(* Logix 5000 project; controller ABB_Drive_Test vendor 1 type 14 code 149 rev 33.12; software revision 33.01 *)

TASK MainTask (continuous, watchdog 500 ms) : T000_MainProgram, CSVProgram, CF_FunctionsProgram

MODULES
   Local : vendor 1 type 14 code 149 (Compact 0, rev 33.12)
      Module_Hart : vendor 58 type 10 code 4 (Compact 2, rev 3.1, Output RPI 80 ms)
      Discrete_IO : Embedded (Compact 1, rev 3.1, Output RPI 20 ms)
      ABBDrive : ETHERNET-MODULE (Ethernet 192.168.2.9, rev 1.1, Output RPI 20 ms)
           ABBDrive:I.Data[0]   // Logic Status Word
           ABBDrive:I.Data[1]   // RPM Actual (INT)
           ABBDrive:I.Data[2]   // DL 1 (Real)
           ABBDrive:I.Data[3]   // DL 1 (Real)
END_MODULES

TYPE ABB_Read :   // Datalinks de Lectura
STRUCT
   Logic_Status_Word : LSW;
   RPM_Feedback : INT;   // RPM Tomada del VSD
   RPM_Referencia : INT;   // Referencia RPM Inyectada
   Output_Power : REAL;
   BusDC : REAL;
   Output_Current : REAL;
   Output_Voltage : REAL;
   PF : REAL;   // Factor de Potencia
   Latest_Fault : INT;
   Accel : BOOL;   // Estado VSD si esta Acelerando
   Descell : BOOL;   // Estado VSD si esta Deshacelerando
END_STRUCT
END_TYPE

TYPE ABB_Write :
STRUCT
   RPM_Reference : INT;
   Run_Forward : BOOL;
   Run_Reverse : BOOL;
   Reset_Fault : BOOL;
END_STRUCT
END_TYPE

TYPE CF_functions :
STRUCT
   command : DINT;   // 1=clear 2=read 3=write 4=append 5=delete 6=rename 7=create dir 8=list 9=list+ 10=list dir 11=detect card 12=get timestamp
   index : DINT;
   offset : DINT;
   REQ_length : DINT;
   DN_length : DINT;
   result : DINT;
   name : STRING;
   newname : STRING;
   data : SINT[460];
   strings : STRING[100];
END_STRUCT
END_TYPE

TYPE ComandVSD :   // Comandos de funcionamiento VSD
STRUCT
   start : BOOL;   // arranque
   stop : BOOL;   // Parada
   reset : BOOL;   // reset VSD
   referencia : REAL;   // Referencia en RPM para VSD AFE
   direction : BOOL;   // Fordware o Reverse
END_STRUCT
END_TYPE

TYPE DateTime :
STRUCT
   year : DINT;
   month : DINT;
   day : DINT;
   hour : DINT;
   minute : DINT;
   second : DINT;
   usec : DINT;
END_STRUCT
END_TYPE

TYPE Dinagrama :   // Estructura de Dinagrama para lectura del SWC PRO
STRUCT
   indiceAux : INT;   // Indice Auxiliar para lectura PLC a SWC
   indice : INT;   // Indice para la lectura del Vector de Potencia
   CT : REAL;   // Valor de la CT para enviar por comunicación a SWC
   PotenciaC : REAL;   // Potencia Cableada valor
   Potencia : REAL;   // Valor de Potencia Actual adquirida por comunicación
   numeroMuestras : INT;   // Numero de Muestras del Stroke de Potencia
   pausa : BOOL;   // Pausa en la adquisión del stroke de potencia
   tiempoMuestreo : INT;   // Tiempo de Muestreo de la señal en ms
   tiempoPausa : INT;   // Tiempo de Pausa para la adquisión de la señal
   vsdActive : BOOL;   // Variador en Referencia
   proximetro : BOOL;   // Señal digital del proximetro tomada de la R003_IO
   inicio : BOOL;   // Inicio para la adquisión de dinagrama, teniendo presente si llego a referencia y demás
   Posicion : REAL;   // Posicion SRP
   Carga : REAL;   // Carga de Sarta Entrada Analoga
   confPos : fuenteEntradaAnaloga;   // Configuracion de Entrada Analoga de posicion
   confCarga : fuenteEntradaAnaloga;   // Configuracion de entrada analoga de carga
   confPot : fuenteEntradaAnaloga;   // Configuracion de entrada analoga VSD
   confCT : fuenteEntradaAnaloga;   // Configuración de Entrada CT
END_STRUCT
END_TYPE

TYPE ethImplicitRead :   // Comunicación para la lectura de los parametros del VSD por ethernet IP
STRUCT
   Enabled : BOOL;   // habilitar Comunicación
   Done : BOOL;   // Se realizó correctamente
   Error : BOOL;   // Se tiene un error en la lectura de los parámetros
   Value : DINT;   // Valor Obtenido
   instance : DINT;   // instancia del parametro
   atribute : INT;   // Atributo del parametro
END_STRUCT
END_TYPE

TYPE ethImplicitWrite :   // Comunicación Para enviar parametros al sistema
STRUCT
   Enabled : BOOL;   // Habilitar
   Done : BOOL;   // Se realizo exitozamente
   ERR : BOOL;   // Error en el envio de la información
   Value : DINT;   // Valor a ingresar
   Instance : DINT;   // Valor de la Instancia
   Atribute : INT;   // Valor del Atributo de la instancia
   clase : INT;
END_STRUCT
END_TYPE

TYPE fuenteEntradaAnaloga :   // Definición de Entrada Analoga ,Fuente de la señal ,rango minimo y maximo
STRUCT
   fuente : INT;   // Canal por el cual se suministra la señal
   Valor : REAL;   // Valor Actual de la señal
   min : REAL;
   max : REAL;
   ValorMinAmp : REAL;
END_STRUCT
END_TYPE

TYPE LSW :   // Drive - Logic Status Word
STRUCT
   Faulted : BOOL;
   Warning : BOOL;
   RunForward : BOOL;
   RunReverse : BOOL;
   Ready : BOOL;
   RemoteRef : BOOL;
   RemoteCrtl : BOOL;
   AtSpeed : BOOL;
END_STRUCT
END_TYPE

TYPE SWC :   // Comunicación Ethernet con el SWC PRO
STRUCT
   comand : ComandVSD;   // Comandos para VSD
   dinagrama : Dinagrama;   // Valores para adquisión del dinagrama
   entradasDigitales : INT;
   salidasDigitales : INT;
   entradasAnalogas : REAL[4];
   salidasAnalogas : REAL[4];
   ABBRead : ABB_Read;   // Valores de Lectura
   etheWrite : ethImplicitWrite;   // Valores de Escritura Ethernet para VSD
   etheRead : ethImplicitRead;   // Valores de Lectura
END_STRUCT
END_TYPE

ADD_ON_INSTRUCTION CF_big_write   (* revision 1.1 *)
// Revision note:
// only act when triggered
VAR_IN_OUT
   command : DINT; {required}
END_VAR
VAR_INPUT
   array_offset : DINT; {required}
END_VAR
VAR_IN_OUT
   CF_ctrl : CF_functions; {required}
   data : SINT[100]; {required}
END_VAR
VAR_OUTPUT
   busy : BOOL; {access Read Only, visible}
END_VAR
VAR
   arsize : DINT;
   stored_req_length : DINT;
   oneshots : DINT;
   bigwrite : BOOL;
   length_diff : DINT;
   bigread : BOOL;
   BW_active : BOOL;
END_VAR

ROUTINE Logic   (* ladder *)
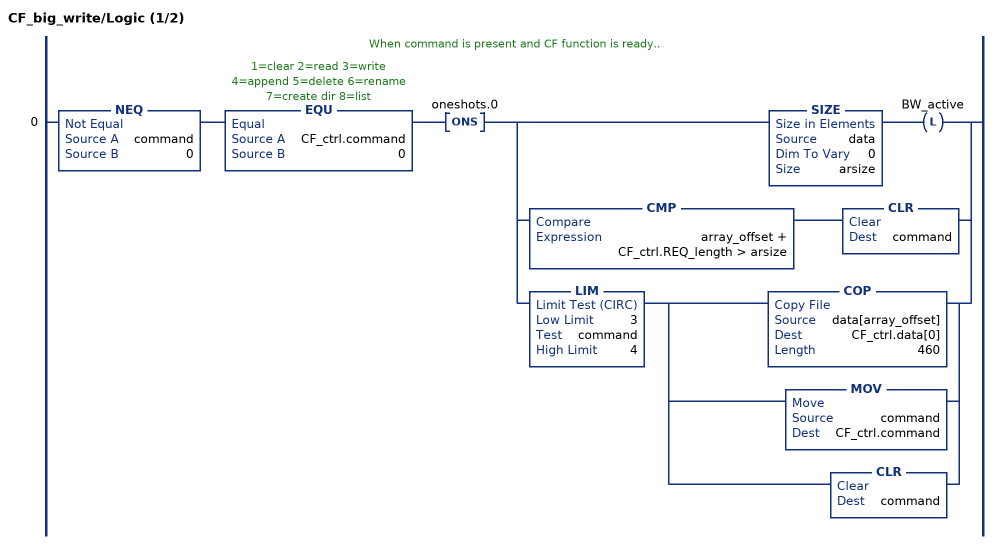
   // When command is present and CF function is ready..
   0: NEQ(command,0)EQU(CF_ctrl.command,0)ONS(oneshots.0)[SIZE(data,0,arsize) OTL(BW_active) ,CMP(array_offset + CF_ctrl.REQ_length > arsize) CLR(command) ,LIM(3,command,4) [COP(data[array_offset],CF_ctrl.data[0],460) ,MOV(command,CF_ctrl.command) ,CLR(command) ] ];
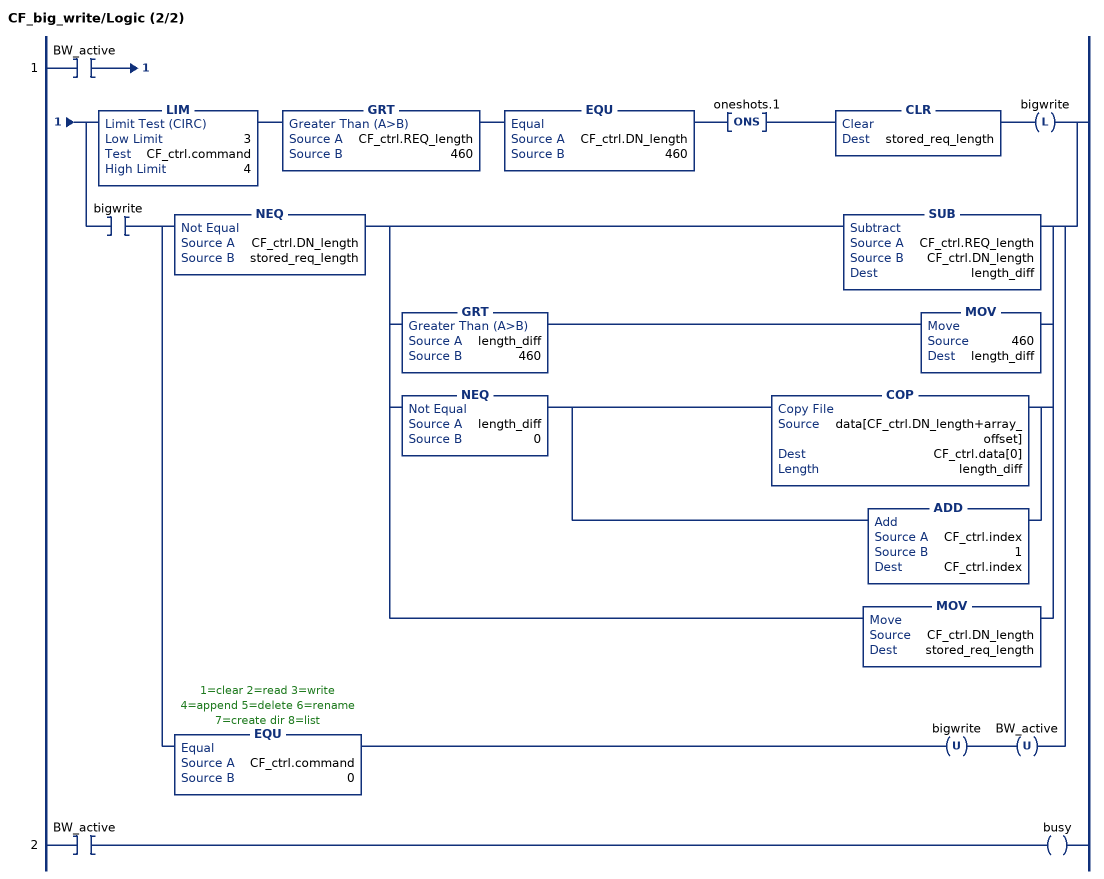
   1: XIC(BW_active)[LIM(3,CF_ctrl.command,4) GRT(CF_ctrl.REQ_length,460) EQU(CF_ctrl.DN_length,460) ONS(oneshots.1) CLR(stored_req_length) OTL(bigwrite) ,XIC(bigwrite) [NEQ(CF_ctrl.DN_length,stored_req_length) [SUB(CF_ctrl.REQ_length,CF_ctrl.DN_length,length_diff) ,GRT(length_diff,460) MOV(460,length_diff) ,NEQ(length_diff,0) [COP(data[CF_ctrl.DN_length+array_offset],CF_ctrl.data[0],length_diff) ,ADD(CF_ctrl.index,1,CF_ctrl.index) ] ,MOV(CF_ctrl.DN_length,stored_req_length) ] ,EQU(CF_ctrl.command,0) OTU(bigwrite) OTU(BW_active) ] ];
   2: XIC(BW_active)OTE(busy);
END_ROUTINE
END_ADD_ON_INSTRUCTION

VAR_GLOBAL   (* controller tags *)
   ABB_GetAtt_Value : DINT := 6000;
   ABB_GetMsg : MESSAGE;
        MessageParameters(ServiceCode := 16#000e, DestinationTag := ABB_GetAtt_Value, ...)
   ABB_Input : ABB_Read := (Logic_Status_Word.Ready := 1, Logic_Status_Word.RemoteRef := 1, Logic_Status_Word.RemoteCrtl := 1, RPM_Referencia := 1440, Output_Power := 5.9449345e-37, BusDC := 678.2, Latest_Fault := 13185);
   ABB_Msg_SetValue : DINT := 1;
   ABB_Output : ABB_Write := (RPM_Reference := 1440);
   ABB_SetMsg : MESSAGE;
        MessageParameters(ServiceCode := 16#0010, LocalElement := ABB_Msg_SetValue, ...)
   asciidata : SINT[11000] := ([0] := 51, [1] := 53, [2] := 56, [3] := 56, [4] := 56, [5] := 44, [6] := 48, [7] := 46, [8] := 48, [9] := 57, [10] := 50, [11] := 55, [12] := 48, [13] := 54, [14] := 54, [15] := 48, [16] := 44, [17] := 50, [18] := 46, [19] := 48, [20] := 48, [21] := 48, [22] := 48, [23] := 48, [24] := 48, [25] := 48, [26] := 48, [27] := 44, [28] := 53, [29] := 46, [30] := 48, [31] := 48, [32] := 48, [33] := 48, [34] := 48, [35] := 48, [36] := 48, [37] := 48, [38] := 44, [39] := 54, [40] := 46, [41] := 48, [42] := 48, [43] := 48, [44] := 48, [45] := 48, [46] := 48, [47] := 48, [48] := 48, [49] := 44, [50] := 55, [51] := 46, [52] := 48, [53] := 48, [54] := 48, [55] := 48, [56] := 48, [57] := 48, [58] := 48, [59] := 48,
        [60] := 44, [61] := 56, [62] := 46, [63] := 48, [64] := 48, [65] := 48, [66] := 48, [67] := 48, [68] := 48, [69] := 48, [70] := 48, [71] := 44, [72] := 57, [73] := 46, [74] := 48, [75] := 48, [76] := 48, [77] := 48, [78] := 48, [79] := 48, [80] := 48, [81] := 48, [82] := 44, [83] := 49, [84] := 48, [85] := 46, [86] := 48, [87] := 48, [88] := 48, [89] := 48, [90] := 48, [91] := 48, [92] := 48, [93] := 44, [94] := 49, [95] := 49, [96] := 46, [97] := 48, [98] := 48, [99] := 48, [100] := 48, [101] := 48, [102] := 48, [103] := 48, [104] := 44, [105] := 49, [106] := 50, [107] := 46, [108] := 48, [109] := 48, [110] := 48, [111] := 48, [112] := 48, [113] := 48, [114] := 48, [115] := 44, [116] := 49, [117] := 46, [118] := 48, [119] := 48,
        [120] := 48, [121] := 48, [122] := 48, [123] := 48, [124] := 48, [125] := 48, [126] := 13, [127] := 10, [128] := 51, [129] := 53, [130] := 56, [131] := 56, [132] := 56, [133] := 44, [134] := 48, [135] := 46, [136] := 48, [137] := 57, [138] := 50, [139] := 55, [140] := 49, [141] := 56, [142] := 49, [143] := 55, [144] := 44, [145] := 50, [146] := 46, [147] := 48, [148] := 48, [149] := 48, [150] := 48, [151] := 48, [152] := 48, [153] := 48, [154] := 48, [155] := 44, [156] := 53, [157] := 46, [158] := 48, [159] := 48, [160] := 48, [161] := 48, [162] := 48, [163] := 48, [164] := 48, [165] := 48, [166] := 44, [167] := 54, [168] := 46, [169] := 48, [170] := 48, [171] := 48, [172] := 48, [173] := 48, [174] := 48, [175] := 48, [176] := 48, [177] := 44, [178] := 55, [179] := 46,
        [180] := 48, [181] := 48, [182] := 48, [183] := 48, [184] := 48, [185] := 48, [186] := 48, [187] := 48, [188] := 44, [189] := 56, [190] := 46, [191] := 48, [192] := 48, [193] := 48, [194] := 48, [195] := 48, [196] := 48, [197] := 48, [198] := 48, [199] := 44, [200] := 57, [201] := 46, [202] := 48, [203] := 48, [204] := 48, [205] := 48, [206] := 48, [207] := 48, [208] := 48, [209] := 48, [210] := 44, [211] := 49, [212] := 48, [213] := 46, [214] := 48, [215] := 48, [216] := 48, [217] := 48, [218] := 48, [219] := 48, [220] := 48, [221] := 44, [222] := 49, [223] := 49, [224] := 46, [225] := 48, [226] := 48, [227] := 48, [228] := 48, [229] := 48, [230] := 48, [231] := 48, [232] := 44, [233] := 49, [234] := 50, [235] := 46, [236] := 48, [237] := 48, [238] := 48, [239] := 48,
        [240] := 48, [241] := 48, [242] := 48, [243] := 44, [244] := 49, [245] := 46, [246] := 48, [247] := 48, [248] := 48, [249] := 48, [250] := 48, [251] := 48, [252] := 48, [253] := 48, [254] := 13, [255] := 10, [256] := 51, [257] := 53, [258] := 56, [259] := 56, [260] := 56, [261] := 44, [262] := 48, [263] := 46, [264] := 48, [265] := 57, [266] := 50, [267] := 55, [268] := 50, [269] := 57, [270] := 55, [271] := 53, [272] := 44, [273] := 50, [274] := 46, [275] := 48, [276] := 48, [277] := 48, [278] := 48, [279] := 48, [280] := 48, [281] := 48, [282] := 48, [283] := 44, [284] := 53, [285] := 46, [286] := 48, [287] := 48, [288] := 48, [289] := 48, [290] := 48, [291] := 48, [292] := 48, [293] := 48, [294] := 44, [295] := 54, [296] := 46, [297] := 48, [298] := 48, [299] := 48,
        [300] := 48, [301] := 48, [302] := 48, [303] := 48, [304] := 48, [305] := 44, [306] := 55, [307] := 46, [308] := 48, [309] := 48, [310] := 48, [311] := 48, [312] := 48, [313] := 48, [314] := 48, [315] := 48, [316] := 44, [317] := 56, [318] := 46, [319] := 48, [320] := 48, [321] := 48, [322] := 48, [323] := 48, [324] := 48, [325] := 48, [326] := 48, [327] := 44, [328] := 57, [329] := 46, [330] := 48, [331] := 48, [332] := 48, [333] := 48, [334] := 48, [335] := 48, [336] := 48, [337] := 48, [338] := 44, [339] := 49, [340] := 48, [341] := 46, [342] := 48, [343] := 48, [344] := 48, [345] := 48, [346] := 48, [347] := 48, [348] := 48, [349] := 44, [350] := 49, [351] := 49, [352] := 46, [353] := 48, [354] := 48, [355] := 48, [356] := 48, [357] := 48, [358] := 48, [359] := 48,
        [360] := 44, [361] := 49, [362] := 50, [363] := 46, [364] := 48, [365] := 48, [366] := 48, [367] := 48, [368] := 48, [369] := 48, [370] := 48, [371] := 44, [372] := 49, [373] := 46, [374] := 48, [375] := 48, [376] := 48, [377] := 48, [378] := 48, [379] := 48, [380] := 48, [381] := 48, [382] := 13, [383] := 10, [384] := 51, [385] := 53, [386] := 56, [387] := 56, [388] := 56, [389] := 44, [390] := 48, [391] := 46, [392] := 48, [393] := 57, [394] := 50, [395] := 55, [396] := 52, [397] := 49, [398] := 51, [399] := 50, [400] := 44, [401] := 50, [402] := 46, [403] := 48, [404] := 48, [405] := 48, [406] := 48, [407] := 48, [408] := 48, [409] := 48, [410] := 48, [411] := 44, [412] := 53, [413] := 46, [414] := 48, [415] := 48, [416] := 48, [417] := 48, [418] := 48, [419] := 48,
        [420] := 48, [421] := 48, [422] := 44, [423] := 54, [424] := 46, [425] := 48, [426] := 48, [427] := 48, [428] := 48, [429] := 48, [430] := 48, [431] := 48, [432] := 48, [433] := 44, [434] := 55, [435] := 46, [436] := 48, [437] := 48, [438] := 48, [439] := 48, [440] := 48, [441] := 48, [442] := 48, [443] := 48, [444] := 44, [445] := 56, [446] := 46, [447] := 48, [448] := 48, [449] := 48, [450] := 48, [451] := 48, [452] := 48, [453] := 48, [454] := 48, [455] := 44, [456] := 57, [457] := 46, [458] := 48, [459] := 48, [460] := 48, [461] := 48, [462] := 48, [463] := 48, [464] := 48, [465] := 48, [466] := 44, [467] := 49, [468] := 48, [469] := 46, [470] := 48, [471] := 48, [472] := 48, [473] := 48, [474] := 48, [475] := 48, [476] := 48, [477] := 44, [478] := 49, [479] := 49,
        [480] := 46, [481] := 48, [482] := 48, [483] := 48, [484] := 48, [485] := 48, [486] := 48, [487] := 48, [488] := 44, [489] := 49, [490] := 50, [491] := 46, [492] := 48, [493] := 48, [494] := 48, [495] := 48, [496] := 48, [497] := 48, [498] := 48, [499] := 44, [500] := 49, [501] := 46, [502] := 48, [503] := 48, [504] := 48, [505] := 48, [506] := 48, [507] := 48, [508] := 48, [509] := 48, [510] := 13, [511] := 10, [512] := 51, [513] := 53, [514] := 56, [515] := 56, [516] := 56, [517] := 44, [518] := 48, [519] := 46, [520] := 48, [521] := 57, [522] := 50, [523] := 55, [524] := 53, [525] := 50, [526] := 57, [527] := 48, [528] := 44, [529] := 50, [530] := 46, [531] := 48, [532] := 48, [533] := 48, [534] := 48, [535] := 48, [536] := 48, [537] := 48, [538] := 48, [539] := 44,
        [540] := 53, [541] := 46, [542] := 48, [543] := 48, [544] := 48, [545] := 48, [546] := 48, [547] := 48, [548] := 48, [549] := 48, [550] := 44, [551] := 54, [552] := 46, [553] := 48, [554] := 48, [555] := 48, [556] := 48, [557] := 48, [558] := 48, [559] := 48, [560] := 48, [561] := 44, [562] := 55, [563] := 46, [564] := 48, [565] := 48, [566] := 48, [567] := 48, [568] := 48, [569] := 48, [570] := 48, [571] := 48, [572] := 44, [573] := 56, [574] := 46, [575] := 48, [576] := 48, [577] := 48, [578] := 48, [579] := 48, [580] := 48, [581] := 48, [582] := 48, [583] := 44, [584] := 57, [585] := 46, [586] := 48, [587] := 48, [588] := 48, [589] := 48, [590] := 48, [591] := 48, [592] := 48, [593] := 48, [594] := 44, [595] := 49, [596] := 48, [597] := 46, [598] := 48, [599] := 48,
        [600] := 48, [601] := 48, [602] := 48, [603] := 48, [604] := 48, [605] := 44, [606] := 49, [607] := 49, [608] := 46, [609] := 48, [610] := 48, [611] := 48, [612] := 48, [613] := 48, [614] := 48, [615] := 48, [616] := 44, [617] := 49, [618] := 50, [619] := 46, [620] := 48, [621] := 48, [622] := 48, [623] := 48, [624] := 48, [625] := 48, [626] := 48, [627] := 44, [628] := 49, [629] := 46, [630] := 48, [631] := 48, [632] := 48, [633] := 48, [634] := 48, [635] := 48, [636] := 48, [637] := 48, [638] := 13, [639] := 10, [640] := 51, [641] := 53, [642] := 56, [643] := 56, [644] := 56, [645] := 44, [646] := 48, [647] := 46, [648] := 48, [649] := 57, [650] := 50, [651] := 55, [652] := 54, [653] := 52, [654] := 52, [655] := 55, [656] := 44, [657] := 50, [658] := 46, [659] := 48,
        [660] := 48, [661] := 48, [662] := 48, [663] := 48, [664] := 48, [665] := 48, [666] := 48, [667] := 44, [668] := 53, [669] := 46, [670] := 48, [671] := 48, [672] := 48, [673] := 48, [674] := 48, [675] := 48, [676] := 48, [677] := 48, [678] := 44, [679] := 54, [680] := 46, [681] := 48, [682] := 48, [683] := 48, [684] := 48, [685] := 48, [686] := 48, [687] := 48, [688] := 48, [689] := 44, [690] := 55, [691] := 46, [692] := 48, [693] := 48, [694] := 48, [695] := 48, [696] := 48, [697] := 48, [698] := 48, [699] := 48, [700] := 44, [701] := 56, [702] := 46, [703] := 48, [704] := 48, [705] := 48, [706] := 48, [707] := 48, [708] := 48, [709] := 48, [710] := 48, [711] := 44, [712] := 57, [713] := 46, [714] := 48, [715] := 48, [716] := 48, [717] := 48, [718] := 48, [719] := 48,
        [720] := 48, [721] := 48, [722] := 44, [723] := 49, [724] := 48, [725] := 46, [726] := 48, [727] := 48, [728] := 48, [729] := 48, [730] := 48, [731] := 48, [732] := 48, [733] := 44, [734] := 49, [735] := 49, [736] := 46, [737] := 48, [738] := 48, [739] := 48, [740] := 48, [741] := 48, [742] := 48, [743] := 48, [744] := 44, [745] := 49, [746] := 50, [747] := 46, [748] := 48, [749] := 48, [750] := 48, [751] := 48, [752] := 48, [753] := 48, [754] := 48, [755] := 44, [756] := 49, [757] := 46, [758] := 48, [759] := 48, [760] := 48, [761] := 48, [762] := 48, [763] := 48, [764] := 48, [765] := 48, [766] := 13, [767] := 10, [768] := 51, [769] := 53, [770] := 56, [771] := 56, [772] := 56, [773] := 44, [774] := 48, [775] := 46, [776] := 48, [777] := 57, [778] := 50, [779] := 55,
        [780] := 55, [781] := 54, [782] := 48, [783] := 53, [784] := 44, [785] := 50, [786] := 46, [787] := 48, [788] := 48, [789] := 48, [790] := 48, [791] := 48, [792] := 48, [793] := 48, [794] := 48, [795] := 44, [796] := 53, [797] := 46, [798] := 48, [799] := 48, [800] := 48, [801] := 48, [802] := 48, [803] := 48, [804] := 48, [805] := 48, [806] := 44, [807] := 54, [808] := 46, [809] := 48, [810] := 48, [811] := 48, [812] := 48, [813] := 48, [814] := 48, [815] := 48, [816] := 48, [817] := 44, [818] := 55, [819] := 46, [820] := 48, [821] := 48, [822] := 48, [823] := 48, [824] := 48, [825] := 48, [826] := 48, [827] := 48, [828] := 44, [829] := 56, [830] := 46, [831] := 48, [832] := 48, [833] := 48, [834] := 48, [835] := 48, [836] := 48, [837] := 48, [838] := 48, [839] := 44,
        [840] := 57, [841] := 46, [842] := 48, [843] := 48, [844] := 48, [845] := 48, [846] := 48, [847] := 48, [848] := 48, [849] := 48, [850] := 44, [851] := 49, [852] := 48, [853] := 46, [854] := 48, [855] := 48, [856] := 48, [857] := 48, [858] := 48, [859] := 48, [860] := 48, [861] := 44, [862] := 49, [863] := 49, [864] := 46, [865] := 48, [866] := 48, [867] := 48, [868] := 48, [869] := 48, [870] := 48, [871] := 48, [872] := 44, [873] := 49, [874] := 50, [875] := 46, [876] := 48, [877] := 48, [878] := 48, [879] := 48, [880] := 48, [881] := 48, [882] := 48, [883] := 44, [884] := 49, [885] := 46, [886] := 48, [887] := 48, [888] := 48, [889] := 48, [890] := 48, [891] := 48, [892] := 48, [893] := 48, [894] := 13, [895] := 10, [896] := 51, [897] := 53, [898] := 56, [899] := 56,
        [900] := 56, [901] := 44, [902] := 48, [903] := 46, [904] := 48, [905] := 57, [906] := 50, [907] := 55, [908] := 56, [909] := 55, [910] := 54, [911] := 50, [912] := 44, [913] := 50, [914] := 46, [915] := 48, [916] := 48, [917] := 48, [918] := 48, [919] := 48, [920] := 48, [921] := 48, [922] := 48, [923] := 44, [924] := 53, [925] := 46, [926] := 48, [927] := 48, [928] := 48, [929] := 48, [930] := 48, [931] := 48, [932] := 48, [933] := 48, [934] := 44, [935] := 54, [936] := 46, [937] := 48, [938] := 48, [939] := 48, [940] := 48, [941] := 48, [942] := 48, [943] := 48, [944] := 48, [945] := 44, [946] := 55, [947] := 46, [948] := 48, [949] := 48, [950] := 48, [951] := 48, [952] := 48, [953] := 48, [954] := 48, [955] := 48, [956] := 44, [957] := 56, [958] := 46, [959] := 48,
        [960] := 48, [961] := 48, [962] := 48, [963] := 48, [964] := 48, [965] := 48, [966] := 48, [967] := 44, [968] := 57, [969] := 46, [970] := 48, [971] := 48, [972] := 48, [973] := 48, [974] := 48, [975] := 48, [976] := 48, [977] := 48, [978] := 44, [979] := 49, [980] := 48, [981] := 46, [982] := 48, [983] := 48, [984] := 48, [985] := 48, [986] := 48, [987] := 48, [988] := 48, [989] := 44, [990] := 49, [991] := 49, [992] := 46, [993] := 48, [994] := 48, [995] := 48, [996] := 48, [997] := 48, [998] := 48, [999] := 48, [1000] := 44, [1001] := 49, [1002] := 50, [1003] := 46, [1004] := 48, [1005] := 48, [1006] := 48, [1007] := 48, [1008] := 48, [1009] := 48, [1010] := 48, [1011] := 44, [1012] := 49, [1013] := 46, [1014] := 48, [1015] := 48, [1016] := 48, [1017] := 48, [1018] := 48, [1019] := 48,
        [1020] := 48, [1021] := 48, [1022] := 13, [1023] := 10, [1024] := 51, [1025] := 53, [1026] := 56, [1027] := 56, [1028] := 56, [1029] := 44, [1030] := 48, [1031] := 46, [1032] := 48, [1033] := 57, [1034] := 50, [1035] := 55, [1036] := 57, [1037] := 57, [1038] := 49, [1039] := 57, [1040] := 44, [1041] := 50, [1042] := 46, [1043] := 48, [1044] := 48, [1045] := 48, [1046] := 48, [1047] := 48, [1048] := 48, [1049] := 48, [1050] := 48, [1051] := 44, [1052] := 53, [1053] := 46, [1054] := 48, [1055] := 48, [1056] := 48, [1057] := 48, [1058] := 48, [1059] := 48, [1060] := 48, [1061] := 48, [1062] := 44, [1063] := 54, [1064] := 46, [1065] := 48, [1066] := 48, [1067] := 48, [1068] := 48, [1069] := 48, [1070] := 48, [1071] := 48, [1072] := 48, [1073] := 44, [1074] := 55, [1075] := 46, [1076] := 48, [1077] := 48, [1078] := 48, [1079] := 48,
        [1080] := 48, [1081] := 48, [1082] := 48, [1083] := 48, [1084] := 44, [1085] := 56, [1086] := 46, [1087] := 48, [1088] := 48, [1089] := 48, [1090] := 48, [1091] := 48, [1092] := 48, [1093] := 48, [1094] := 48, [1095] := 44, [1096] := 57, [1097] := 46, [1098] := 48, [1099] := 48, [1100] := 48, [1101] := 48, [1102] := 48, [1103] := 48, [1104] := 48, [1105] := 48, [1106] := 44, [1107] := 49, [1108] := 48, [1109] := 46, [1110] := 48, [1111] := 48, [1112] := 48, [1113] := 48, [1114] := 48, [1115] := 48, [1116] := 48, [1117] := 44, [1118] := 49, [1119] := 49, [1120] := 46, [1121] := 48, [1122] := 48, [1123] := 48, [1124] := 48, [1125] := 48, [1126] := 48, [1127] := 48, [1128] := 44, [1129] := 49, [1130] := 50, [1131] := 46, [1132] := 48, [1133] := 48, [1134] := 48, [1135] := 48, [1136] := 48, [1137] := 48, [1138] := 48, [1139] := 44,
        [1140] := 49, [1141] := 46, [1142] := 48, [1143] := 48, [1144] := 48, [1145] := 48, [1146] := 48, [1147] := 48, [1148] := 48, [1149] := 48, [1150] := 13, [1151] := 10, [1152] := 51, [1153] := 53, [1154] := 56, [1155] := 56, [1156] := 56, [1157] := 44, [1158] := 48, [1159] := 46, [1160] := 48, [1161] := 57, [1162] := 50, [1163] := 56, [1164] := 49, [1165] := 48, [1166] := 55, [1167] := 54, [1168] := 44, [1169] := 50, [1170] := 46, [1171] := 48, [1172] := 48, [1173] := 48, [1174] := 48, [1175] := 48, [1176] := 48, [1177] := 48, [1178] := 48, [1179] := 44, [1180] := 53, [1181] := 46, [1182] := 48, [1183] := 48, [1184] := 48, [1185] := 48, [1186] := 48, [1187] := 48, [1188] := 48, [1189] := 48, [1190] := 44, [1191] := 54, [1192] := 46, [1193] := 48, [1194] := 48, [1195] := 48, [1196] := 48, [1197] := 48, [1198] := 48, [1199] := 48,
        [1200] := 48, [1201] := 44, [1202] := 55, [1203] := 46, [1204] := 48, [1205] := 48, [1206] := 48, [1207] := 48, [1208] := 48, [1209] := 48, [1210] := 48, [1211] := 48, [1212] := 44, [1213] := 56, [1214] := 46, [1215] := 48, [1216] := 48, [1217] := 48, [1218] := 48, [1219] := 48, [1220] := 48, [1221] := 48, [1222] := 48, [1223] := 44, [1224] := 57, [1225] := 46, [1226] := 48, [1227] := 48, [1228] := 48, [1229] := 48, [1230] := 48, [1231] := 48, [1232] := 48, [1233] := 48, [1234] := 44, [1235] := 49, [1236] := 48, [1237] := 46, [1238] := 48, [1239] := 48, [1240] := 48, [1241] := 48, [1242] := 48, [1243] := 48, [1244] := 48, [1245] := 44, [1246] := 49, [1247] := 49, [1248] := 46, [1249] := 48, [1250] := 48, [1251] := 48, [1252] := 48, [1253] := 48, [1254] := 48, [1255] := 48, [1256] := 44, [1257] := 49, [1258] := 50, [1259] := 46,
        [1260] := 48, [1261] := 48, [1262] := 48, [1263] := 48, [1264] := 48, [1265] := 48, [1266] := 48, [1267] := 44, [1268] := 49, [1269] := 46, [1270] := 48, [1271] := 48, [1272] := 48, [1273] := 48, [1274] := 48, [1275] := 48, [1276] := 48, [1277] := 48, [1278] := 13, [1279] := 10, [1280] := 51, [1281] := 53, [1282] := 56, [1283] := 56, [1284] := 56, [1285] := 44, [1286] := 48, [1287] := 46, [1288] := 48, [1289] := 57, [1290] := 50, [1291] := 56, [1292] := 50, [1293] := 50, [1294] := 51, [1295] := 52, [1296] := 44, [1297] := 50, [1298] := 46, [1299] := 48, [1300] := 48, [1301] := 48, [1302] := 48, [1303] := 48, [1304] := 48, [1305] := 48, [1306] := 48, [1307] := 44, [1308] := 53, [1309] := 46, [1310] := 48, [1311] := 48, [1312] := 48, [1313] := 48, [1314] := 48, [1315] := 48, [1316] := 48, [1317] := 48, [1318] := 44, [1319] := 54,
        [1320] := 46, [1321] := 48, [1322] := 48, [1323] := 48, [1324] := 48, [1325] := 48, [1326] := 48, [1327] := 48, [1328] := 48, [1329] := 44, [1330] := 55, [1331] := 46, [1332] := 48, [1333] := 48, [1334] := 48, [1335] := 48, [1336] := 48, [1337] := 48, [1338] := 48, [1339] := 48, [1340] := 44, [1341] := 56, [1342] := 46, [1343] := 48, [1344] := 48, [1345] := 48, [1346] := 48, [1347] := 48, [1348] := 48, [1349] := 48, [1350] := 48, [1351] := 44, [1352] := 57, [1353] := 46, [1354] := 48, [1355] := 48, [1356] := 48, [1357] := 48, [1358] := 48, [1359] := 48, [1360] := 48, [1361] := 48, [1362] := 44, [1363] := 49, [1364] := 48, [1365] := 46, [1366] := 48, [1367] := 48, [1368] := 48, [1369] := 48, [1370] := 48, [1371] := 48, [1372] := 48, [1373] := 44, [1374] := 49, [1375] := 49, [1376] := 46, [1377] := 48, [1378] := 48, [1379] := 48,
        [1380] := 48, [1381] := 48, [1382] := 48, [1383] := 48, [1384] := 44, [1385] := 49, [1386] := 50, [1387] := 46, [1388] := 48, [1389] := 48, [1390] := 48, [1391] := 48, [1392] := 48, [1393] := 48, [1394] := 48, [1395] := 44, [1396] := 49, [1397] := 46, [1398] := 48, [1399] := 48, [1400] := 48, [1401] := 48, [1402] := 48, [1403] := 48, [1404] := 48, [1405] := 48, [1406] := 13, [1407] := 10, [1408] := 51, [1409] := 53, [1410] := 56, [1411] := 56, [1412] := 56, [1413] := 44, [1414] := 48, [1415] := 46, [1416] := 48, [1417] := 57, [1418] := 50, [1419] := 56, [1420] := 51, [1421] := 51, [1422] := 57, [1423] := 49, [1424] := 44, [1425] := 50, [1426] := 46, [1427] := 48, [1428] := 48, [1429] := 48, [1430] := 48, [1431] := 48, [1432] := 48, [1433] := 48, [1434] := 48, [1435] := 44, [1436] := 53, [1437] := 46, [1438] := 48, [1439] := 48,
        [1440] := 48, [1441] := 48, [1442] := 48, [1443] := 48, [1444] := 48, [1445] := 48, [1446] := 44, [1447] := 54, [1448] := 46, [1449] := 48, [1450] := 48, [1451] := 48, [1452] := 48, [1453] := 48, [1454] := 48, [1455] := 48, [1456] := 48, [1457] := 44, [1458] := 55, [1459] := 46, [1460] := 48, [1461] := 48, [1462] := 48, [1463] := 48, [1464] := 48, [1465] := 48, [1466] := 48, [1467] := 48, [1468] := 44, [1469] := 56, [1470] := 46, [1471] := 48, [1472] := 48, [1473] := 48, [1474] := 48, [1475] := 48, [1476] := 48, [1477] := 48, [1478] := 48, [1479] := 44, [1480] := 57, [1481] := 46, [1482] := 48, [1483] := 48, [1484] := 48, [1485] := 48, [1486] := 48, [1487] := 48, [1488] := 48, [1489] := 48, [1490] := 44, [1491] := 49, [1492] := 48, [1493] := 46, [1494] := 48, [1495] := 48, [1496] := 48, [1497] := 48, [1498] := 48, [1499] := 48,
        [1500] := 48, [1501] := 44, [1502] := 49, [1503] := 49, [1504] := 46, [1505] := 48, [1506] := 48, [1507] := 48, [1508] := 48, [1509] := 48, [1510] := 48, [1511] := 48, [1512] := 44, [1513] := 49, [1514] := 50, [1515] := 46, [1516] := 48, [1517] := 48, [1518] := 48, [1519] := 48, [1520] := 48, [1521] := 48, [1522] := 48, [1523] := 44, [1524] := 49, [1525] := 46, [1526] := 48, [1527] := 48, [1528] := 48, [1529] := 48, [1530] := 48, [1531] := 48, [1532] := 48, [1533] := 48, [1534] := 13, [1535] := 10, [1536] := 51, [1537] := 53, [1538] := 56, [1539] := 56, [1540] := 56, [1541] := 44, [1542] := 48, [1543] := 46, [1544] := 48, [1545] := 57, [1546] := 50, [1547] := 56, [1548] := 52, [1549] := 53, [1550] := 52, [1551] := 56, [1552] := 44, [1553] := 50, [1554] := 46, [1555] := 48, [1556] := 48, [1557] := 48, [1558] := 48, [1559] := 48,
        [1560] := 48, [1561] := 48, [1562] := 48, [1563] := 44, [1564] := 53, [1565] := 46, [1566] := 48, [1567] := 48, [1568] := 48, [1569] := 48, [1570] := 48, [1571] := 48, [1572] := 48, [1573] := 48, [1574] := 44, [1575] := 54, [1576] := 46, [1577] := 48, [1578] := 48, [1579] := 48, [1580] := 48, [1581] := 48, [1582] := 48, [1583] := 48, [1584] := 48, [1585] := 44, [1586] := 55, [1587] := 46, [1588] := 48, [1589] := 48, [1590] := 48, [1591] := 48, [1592] := 48, [1593] := 48, [1594] := 48, [1595] := 48, [1596] := 44, [1597] := 56, [1598] := 46, [1599] := 48, [1600] := 48, [1601] := 48, [1602] := 48, [1603] := 48, [1604] := 48, [1605] := 48, [1606] := 48, [1607] := 44, [1608] := 57, [1609] := 46, [1610] := 48, [1611] := 48, [1612] := 48, [1613] := 48, [1614] := 48, [1615] := 48, [1616] := 48, [1617] := 48, [1618] := 44, [1619] := 49,
        [1620] := 48, [1621] := 46, [1622] := 48, [1623] := 48, [1624] := 48, [1625] := 48, [1626] := 48, [1627] := 48, [1628] := 48, [1629] := 44, [1630] := 49, [1631] := 49, [1632] := 46, [1633] := 48, [1634] := 48, [1635] := 48, [1636] := 48, [1637] := 48, [1638] := 48, [1639] := 48, [1640] := 44, [1641] := 49, [1642] := 50, [1643] := 46, [1644] := 48, [1645] := 48, [1646] := 48, [1647] := 48, [1648] := 48, [1649] := 48, [1650] := 48, [1651] := 44, [1652] := 49, [1653] := 46, [1654] := 48, [1655] := 48, [1656] := 48, [1657] := 48, [1658] := 48, [1659] := 48, [1660] := 48, [1661] := 48, [1662] := 13, [1663] := 10, [1664] := 51, [1665] := 53, [1666] := 56, [1667] := 56, [1668] := 56, [1669] := 44, [1670] := 48, [1671] := 46, [1672] := 48, [1673] := 57, [1674] := 50, [1675] := 56, [1676] := 53, [1677] := 55, [1678] := 48, [1679] := 54,
        [1680] := 44, [1681] := 50, [1682] := 46, [1683] := 48, [1684] := 48, [1685] := 48, [1686] := 48, [1687] := 48, [1688] := 48, [1689] := 48, [1690] := 48, [1691] := 44, [1692] := 53, [1693] := 46, [1694] := 48, [1695] := 48, [1696] := 48, [1697] := 48, [1698] := 48, [1699] := 48, [1700] := 48, [1701] := 48, [1702] := 44, [1703] := 54, [1704] := 46, [1705] := 48, [1706] := 48, [1707] := 48, [1708] := 48, [1709] := 48, [1710] := 48, [1711] := 48, [1712] := 48, [1713] := 44, [1714] := 55, [1715] := 46, [1716] := 48, [1717] := 48, [1718] := 48, [1719] := 48, [1720] := 48, [1721] := 48, [1722] := 48, [1723] := 48, [1724] := 44, [1725] := 56, [1726] := 46, [1727] := 48, [1728] := 48, [1729] := 48, [1730] := 48, [1731] := 48, [1732] := 48, [1733] := 48, [1734] := 48, [1735] := 44, [1736] := 57, [1737] := 46, [1738] := 48, [1739] := 48,
        [1740] := 48, [1741] := 48, [1742] := 48, [1743] := 48, [1744] := 48, [1745] := 48, [1746] := 44, [1747] := 49, [1748] := 48, [1749] := 46, [1750] := 48, [1751] := 48, [1752] := 48, [1753] := 48, [1754] := 48, [1755] := 48, [1756] := 48, [1757] := 44, [1758] := 49, [1759] := 49, [1760] := 46, [1761] := 48, [1762] := 48, [1763] := 48, [1764] := 48, [1765] := 48, [1766] := 48, [1767] := 48, [1768] := 44, [1769] := 49, [1770] := 50, [1771] := 46, [1772] := 48, [1773] := 48, [1774] := 48, [1775] := 48, [1776] := 48, [1777] := 48, [1778] := 48, [1779] := 44, [1780] := 49, [1781] := 46, [1782] := 48, [1783] := 48, [1784] := 48, [1785] := 48, [1786] := 48, [1787] := 48, [1788] := 48, [1789] := 48, [1790] := 13, [1791] := 10, [1792] := 51, [1793] := 53, [1794] := 56, [1795] := 56, [1796] := 56, [1797] := 44, [1798] := 48, [1799] := 46,
        [1800] := 48, [1801] := 57, [1802] := 50, [1803] := 56, [1804] := 54, [1805] := 56, [1806] := 54, [1807] := 51, [1808] := 44, [1809] := 50, [1810] := 46, [1811] := 48, [1812] := 48, [1813] := 48, [1814] := 48, [1815] := 48, [1816] := 48, [1817] := 48, [1818] := 48, [1819] := 44, [1820] := 53, [1821] := 46, [1822] := 48, [1823] := 48, [1824] := 48, [1825] := 48, [1826] := 48, [1827] := 48, [1828] := 48, [1829] := 48, [1830] := 44, [1831] := 54, [1832] := 46, [1833] := 48, [1834] := 48, [1835] := 48, [1836] := 48, [1837] := 48, [1838] := 48, [1839] := 48, [1840] := 48, [1841] := 44, [1842] := 55, [1843] := 46, [1844] := 48, [1845] := 48, [1846] := 48, [1847] := 48, [1848] := 48, [1849] := 48, [1850] := 48, [1851] := 48, [1852] := 44, [1853] := 56, [1854] := 46, [1855] := 48, [1856] := 48, [1857] := 48, [1858] := 48, [1859] := 48,
        [1860] := 48, [1861] := 48, [1862] := 48, [1863] := 44, [1864] := 57, [1865] := 46, [1866] := 48, [1867] := 48, [1868] := 48, [1869] := 48, [1870] := 48, [1871] := 48, [1872] := 48, [1873] := 48, [1874] := 44, [1875] := 49, [1876] := 48, [1877] := 46, [1878] := 48, [1879] := 48, [1880] := 48, [1881] := 48, [1882] := 48, [1883] := 48, [1884] := 48, [1885] := 44, [1886] := 49, [1887] := 49, [1888] := 46, [1889] := 48, [1890] := 48, [1891] := 48, [1892] := 48, [1893] := 48, [1894] := 48, [1895] := 48, [1896] := 44, [1897] := 49, [1898] := 50, [1899] := 46, [1900] := 48, [1901] := 48, [1902] := 48, [1903] := 48, [1904] := 48, [1905] := 48, [1906] := 48, [1907] := 44, [1908] := 49, [1909] := 46, [1910] := 48, [1911] := 48, [1912] := 48, [1913] := 48, [1914] := 48, [1915] := 48, [1916] := 48, [1917] := 48, [1918] := 13, [1919] := 10,
        [1920] := 51, [1921] := 53, [1922] := 56, [1923] := 56, [1924] := 56, [1925] := 44, [1926] := 48, [1927] := 46, [1928] := 48, [1929] := 57, [1930] := 50, [1931] := 56, [1932] := 56, [1933] := 48, [1934] := 50, [1935] := 49, [1936] := 44, [1937] := 50, [1938] := 46, [1939] := 48, [1940] := 48, [1941] := 48, [1942] := 48, [1943] := 48, [1944] := 48, [1945] := 48, [1946] := 48, [1947] := 44, [1948] := 53, [1949] := 46, [1950] := 48, [1951] := 48, [1952] := 48, [1953] := 48, [1954] := 48, [1955] := 48, [1956] := 48, [1957] := 48, [1958] := 44, [1959] := 54, [1960] := 46, [1961] := 48, [1962] := 48, [1963] := 48, [1964] := 48, [1965] := 48, [1966] := 48, [1967] := 48, [1968] := 48, [1969] := 44, [1970] := 55, [1971] := 46, [1972] := 48, [1973] := 48, [1974] := 48, [1975] := 48, [1976] := 48, [1977] := 48, [1978] := 48, [1979] := 48,
        [1980] := 44, [1981] := 56, [1982] := 46, [1983] := 48, [1984] := 48, [1985] := 48, [1986] := 48, [1987] := 48, [1988] := 48, [1989] := 48, [1990] := 48, [1991] := 44, [1992] := 57, [1993] := 46, [1994] := 48, [1995] := 48, [1996] := 48, [1997] := 48, [1998] := 48, [1999] := 48, [2000] := 48, [2001] := 48, [2002] := 44, [2003] := 49, [2004] := 48, [2005] := 46, [2006] := 48, [2007] := 48, [2008] := 48, [2009] := 48, [2010] := 48, [2011] := 48, [2012] := 48, [2013] := 44, [2014] := 49, [2015] := 49, [2016] := 46, [2017] := 48, [2018] := 48, [2019] := 48, [2020] := 48, [2021] := 48, [2022] := 48, [2023] := 48, [2024] := 44, [2025] := 49, [2026] := 50, [2027] := 46, [2028] := 48, [2029] := 48, [2030] := 48, [2031] := 48, [2032] := 48, [2033] := 48, [2034] := 48, [2035] := 44, [2036] := 49, [2037] := 46, [2038] := 48, [2039] := 48,
        [2040] := 48, [2041] := 48, [2042] := 48, [2043] := 48, [2044] := 48, [2045] := 48, [2046] := 13, [2047] := 10, [2048] := 51, [2049] := 53, [2050] := 56, [2051] := 56, [2052] := 56, [2053] := 44, [2054] := 48, [2055] := 46, [2056] := 48, [2057] := 57, [2058] := 50, [2059] := 56, [2060] := 57, [2061] := 49, [2062] := 55, [2063] := 56, [2064] := 44, [2065] := 50, [2066] := 46, [2067] := 48, [2068] := 48, [2069] := 48, [2070] := 48, [2071] := 48, [2072] := 48, [2073] := 48, [2074] := 48, [2075] := 44, [2076] := 53, [2077] := 46, [2078] := 48, [2079] := 48, [2080] := 48, [2081] := 48, [2082] := 48, [2083] := 48, [2084] := 48, [2085] := 48, [2086] := 44, [2087] := 54, [2088] := 46, [2089] := 48, [2090] := 48, [2091] := 48, [2092] := 48, [2093] := 48, [2094] := 48, [2095] := 48, [2096] := 48, [2097] := 44, [2098] := 55, [2099] := 46,
        [2100] := 48, [2101] := 48, [2102] := 48, [2103] := 48, [2104] := 48, [2105] := 48, [2106] := 48, [2107] := 48, [2108] := 44, [2109] := 56, [2110] := 46, [2111] := 48, [2112] := 48, [2113] := 48, [2114] := 48, [2115] := 48, [2116] := 48, [2117] := 48, [2118] := 48, [2119] := 44, [2120] := 57, [2121] := 46, [2122] := 48, [2123] := 48, [2124] := 48, [2125] := 48, [2126] := 48, [2127] := 48, [2128] := 48, [2129] := 48, [2130] := 44, [2131] := 49, [2132] := 48, [2133] := 46, [2134] := 48, [2135] := 48, [2136] := 48, [2137] := 48, [2138] := 48, [2139] := 48, [2140] := 48, [2141] := 44, [2142] := 49, [2143] := 49, [2144] := 46, [2145] := 48, [2146] := 48, [2147] := 48, [2148] := 48, [2149] := 48, [2150] := 48, [2151] := 48, [2152] := 44, [2153] := 49, [2154] := 50, [2155] := 46, [2156] := 48, [2157] := 48, [2158] := 48, [2159] := 48,
        [2160] := 48, [2161] := 48, [2162] := 48, [2163] := 44, [2164] := 49, [2165] := 46, [2166] := 48, [2167] := 48, [2168] := 48, [2169] := 48, [2170] := 48, [2171] := 48, [2172] := 48, [2173] := 48, [2174] := 13, [2175] := 10, [2176] := 51, [2177] := 53, [2178] := 56, [2179] := 56, [2180] := 56, [2181] := 44, [2182] := 48, [2183] := 46, [2184] := 48, [2185] := 57, [2186] := 50, [2187] := 57, [2188] := 48, [2189] := 51, [2190] := 51, [2191] := 53, [2192] := 44, [2193] := 50, [2194] := 46, [2195] := 48, [2196] := 48, [2197] := 48, [2198] := 48, [2199] := 48, [2200] := 48, [2201] := 48, [2202] := 48, [2203] := 44, [2204] := 53, [2205] := 46, [2206] := 48, [2207] := 48, [2208] := 48, [2209] := 48, [2210] := 48, [2211] := 48, [2212] := 48, [2213] := 48, [2214] := 44, [2215] := 54, [2216] := 46, [2217] := 48, [2218] := 48, [2219] := 48,
        [2220] := 48, [2221] := 48, [2222] := 48, [2223] := 48, [2224] := 48, [2225] := 44, [2226] := 55, [2227] := 46, [2228] := 48, [2229] := 48, [2230] := 48, [2231] := 48, [2232] := 48, [2233] := 48, [2234] := 48, [2235] := 48, [2236] := 44, [2237] := 56, [2238] := 46, [2239] := 48, [2240] := 48, [2241] := 48, [2242] := 48, [2243] := 48, [2244] := 48, [2245] := 48, [2246] := 48, [2247] := 44, [2248] := 57, [2249] := 46, [2250] := 48, [2251] := 48, [2252] := 48, [2253] := 48, [2254] := 48, [2255] := 48, [2256] := 48, [2257] := 48, [2258] := 44, [2259] := 49, [2260] := 48, [2261] := 46, [2262] := 48, [2263] := 48, [2264] := 48, [2265] := 48, [2266] := 48, [2267] := 48, [2268] := 48, [2269] := 44, [2270] := 49, [2271] := 49, [2272] := 46, [2273] := 48, [2274] := 48, [2275] := 48, [2276] := 48, [2277] := 48, [2278] := 48, [2279] := 48,
        [2280] := 44, [2281] := 49, [2282] := 50, [2283] := 46, [2284] := 48, [2285] := 48, [2286] := 48, [2287] := 48, [2288] := 48, [2289] := 48, [2290] := 48, [2291] := 44, [2292] := 49, [2293] := 46, [2294] := 48, [2295] := 48, [2296] := 48, [2297] := 48, [2298] := 48, [2299] := 48, [2300] := 48, [2301] := 48, [2302] := 13, [2303] := 10, [2304] := 51, [2305] := 53, [2306] := 56, [2307] := 56, [2308] := 56, [2309] := 44, [2310] := 48, [2311] := 46, [2312] := 48, [2313] := 57, [2314] := 50, [2315] := 57, [2316] := 49, [2317] := 52, [2318] := 57, [2319] := 51, [2320] := 44, [2321] := 50, [2322] := 46, [2323] := 48, [2324] := 48, [2325] := 48, [2326] := 48, [2327] := 48, [2328] := 48, [2329] := 48, [2330] := 48, [2331] := 44, [2332] := 53, [2333] := 46, [2334] := 48, [2335] := 48, [2336] := 48, [2337] := 48, [2338] := 48, [2339] := 48,
        [2340] := 48, [2341] := 48, [2342] := 44, [2343] := 54, [2344] := 46, [2345] := 48, [2346] := 48, [2347] := 48, [2348] := 48, [2349] := 48, [2350] := 48, [2351] := 48, [2352] := 48, [2353] := 44, [2354] := 55, [2355] := 46, [2356] := 48, [2357] := 48, [2358] := 48, [2359] := 48, [2360] := 48, [2361] := 48, [2362] := 48, [2363] := 48, [2364] := 44, [2365] := 56, [2366] := 46, [2367] := 48, [2368] := 48, [2369] := 48, [2370] := 48, [2371] := 48, [2372] := 48, [2373] := 48, [2374] := 48, [2375] := 44, [2376] := 57, [2377] := 46, [2378] := 48, [2379] := 48, [2380] := 48, [2381] := 48, [2382] := 48, [2383] := 48, [2384] := 48, [2385] := 48, [2386] := 44, [2387] := 49, [2388] := 48, [2389] := 46, [2390] := 48, [2391] := 48, [2392] := 48, [2393] := 48, [2394] := 48, [2395] := 48, [2396] := 48, [2397] := 44, [2398] := 49, [2399] := 49,
        [2400] := 46, [2401] := 48, [2402] := 48, [2403] := 48, [2404] := 48, [2405] := 48, [2406] := 48, [2407] := 48, [2408] := 44, [2409] := 49, [2410] := 50, [2411] := 46, [2412] := 48, [2413] := 48, [2414] := 48, [2415] := 48, [2416] := 48, [2417] := 48, [2418] := 48, [2419] := 44, [2420] := 49, [2421] := 46, [2422] := 48, [2423] := 48, [2424] := 48, [2425] := 48, [2426] := 48, [2427] := 48, [2428] := 48, [2429] := 48, [2430] := 13, [2431] := 10, [2432] := 51, [2433] := 53, [2434] := 56, [2435] := 56, [2436] := 56, [2437] := 44, [2438] := 48, [2439] := 46, [2440] := 48, [2441] := 57, [2442] := 50, [2443] := 57, [2444] := 50, [2445] := 54, [2446] := 53, [2447] := 48, [2448] := 44, [2449] := 50, [2450] := 46, [2451] := 48, [2452] := 48, [2453] := 48, [2454] := 48, [2455] := 48, [2456] := 48, [2457] := 48, [2458] := 48, [2459] := 44,
        [2460] := 53, [2461] := 46, [2462] := 48, [2463] := 48, [2464] := 48, [2465] := 48, [2466] := 48, [2467] := 48, [2468] := 48, [2469] := 48, [2470] := 44, [2471] := 54, [2472] := 46, [2473] := 48, [2474] := 48, [2475] := 48, [2476] := 48, [2477] := 48, [2478] := 48, [2479] := 48, [2480] := 48, [2481] := 44, [2482] := 55, [2483] := 46, [2484] := 48, [2485] := 48, [2486] := 48, [2487] := 48, [2488] := 48, [2489] := 48, [2490] := 48, [2491] := 48, [2492] := 44, [2493] := 56, [2494] := 46, [2495] := 48, [2496] := 48, [2497] := 48, [2498] := 48, [2499] := 48, [2500] := 48, [2501] := 48, [2502] := 48, [2503] := 44, [2504] := 57, [2505] := 46, [2506] := 48, [2507] := 48, [2508] := 48, [2509] := 48, [2510] := 48, [2511] := 48, [2512] := 48, [2513] := 48, [2514] := 44, [2515] := 49, [2516] := 48, [2517] := 46, [2518] := 48, [2519] := 48,
        [2520] := 48, [2521] := 48, [2522] := 48, [2523] := 48, [2524] := 48, [2525] := 44, [2526] := 49, [2527] := 49, [2528] := 46, [2529] := 48, [2530] := 48, [2531] := 48, [2532] := 48, [2533] := 48, [2534] := 48, [2535] := 48, [2536] := 44, [2537] := 49, [2538] := 50, [2539] := 46, [2540] := 48, [2541] := 48, [2542] := 48, [2543] := 48, [2544] := 48, [2545] := 48, [2546] := 48, [2547] := 44, [2548] := 49, [2549] := 46, [2550] := 48, [2551] := 48, [2552] := 48, [2553] := 48, [2554] := 48, [2555] := 48, [2556] := 48, [2557] := 48, [2558] := 13, [2559] := 10, [2560] := 51, [2561] := 53, [2562] := 56, [2563] := 56, [2564] := 56, [2565] := 44, [2566] := 48, [2567] := 46, [2568] := 48, [2569] := 57, [2570] := 50, [2571] := 57, [2572] := 51, [2573] := 56, [2574] := 48, [2575] := 55, [2576] := 44, [2577] := 50, [2578] := 46, [2579] := 48,
        [2580] := 48, [2581] := 48, [2582] := 48, [2583] := 48, [2584] := 48, [2585] := 48, [2586] := 48, [2587] := 44, [2588] := 53, [2589] := 46, [2590] := 48, [2591] := 48, [2592] := 48, [2593] := 48, [2594] := 48, [2595] := 48, [2596] := 48, [2597] := 48, [2598] := 44, [2599] := 54, [2600] := 46, [2601] := 48, [2602] := 48, [2603] := 48, [2604] := 48, [2605] := 48, [2606] := 48, [2607] := 48, [2608] := 48, [2609] := 44, [2610] := 55, [2611] := 46, [2612] := 48, [2613] := 48, [2614] := 48, [2615] := 48, [2616] := 48, [2617] := 48, [2618] := 48, [2619] := 48, [2620] := 44, [2621] := 56, [2622] := 46, [2623] := 48, [2624] := 48, [2625] := 48, [2626] := 48, [2627] := 48, [2628] := 48, [2629] := 48, [2630] := 48, [2631] := 44, [2632] := 57, [2633] := 46, [2634] := 48, [2635] := 48, [2636] := 48, [2637] := 48, [2638] := 48, [2639] := 48,
        [2640] := 48, [2641] := 48, [2642] := 44, [2643] := 49, [2644] := 48, [2645] := 46, [2646] := 48, [2647] := 48, [2648] := 48, [2649] := 48, [2650] := 48, [2651] := 48, [2652] := 48, [2653] := 44, [2654] := 49, [2655] := 49, [2656] := 46, [2657] := 48, [2658] := 48, [2659] := 48, [2660] := 48, [2661] := 48, [2662] := 48, [2663] := 48, [2664] := 44, [2665] := 49, [2666] := 50, [2667] := 46, [2668] := 48, [2669] := 48, [2670] := 48, [2671] := 48, [2672] := 48, [2673] := 48, [2674] := 48, [2675] := 44, [2676] := 49, [2677] := 46, [2678] := 48, [2679] := 48, [2680] := 48, [2681] := 48, [2682] := 48, [2683] := 48, [2684] := 48, [2685] := 48, [2686] := 13, [2687] := 10, [2688] := 51, [2689] := 53, [2690] := 56, [2691] := 56, [2692] := 56, [2693] := 44, [2694] := 48, [2695] := 46, [2696] := 48, [2697] := 57, [2698] := 50, [2699] := 57,
        [2700] := 52, [2701] := 57, [2702] := 54, [2703] := 53, [2704] := 44, [2705] := 50, [2706] := 46, [2707] := 48, [2708] := 48, [2709] := 48, [2710] := 48, [2711] := 48, [2712] := 48, [2713] := 48, [2714] := 48, [2715] := 44, [2716] := 53, [2717] := 46, [2718] := 48, [2719] := 48, [2720] := 48, [2721] := 48, [2722] := 48, [2723] := 48, [2724] := 48, [2725] := 48, [2726] := 44, [2727] := 54, [2728] := 46, [2729] := 48, [2730] := 48, [2731] := 48, [2732] := 48, [2733] := 48, [2734] := 48, [2735] := 48, [2736] := 48, [2737] := 44, [2738] := 55, [2739] := 46, [2740] := 48, [2741] := 48, [2742] := 48, [2743] := 48, [2744] := 48, [2745] := 48, [2746] := 48, [2747] := 48, [2748] := 44, [2749] := 56, [2750] := 46, [2751] := 48, [2752] := 48, [2753] := 48, [2754] := 48, [2755] := 48, [2756] := 48, [2757] := 48, [2758] := 48, [2759] := 44,
        [2760] := 57, [2761] := 46, [2762] := 48, [2763] := 48, [2764] := 48, [2765] := 48, [2766] := 48, [2767] := 48, [2768] := 48, [2769] := 48, [2770] := 44, [2771] := 49, [2772] := 48, [2773] := 46, [2774] := 48, [2775] := 48, [2776] := 48, [2777] := 48, [2778] := 48, [2779] := 48, [2780] := 48, [2781] := 44, [2782] := 49, [2783] := 49, [2784] := 46, [2785] := 48, [2786] := 48, [2787] := 48, [2788] := 48, [2789] := 48, [2790] := 48, [2791] := 48, [2792] := 44, [2793] := 49, [2794] := 50, [2795] := 46, [2796] := 48, [2797] := 48, [2798] := 48, [2799] := 48, [2800] := 48, [2801] := 48, [2802] := 48, [2803] := 44, [2804] := 49, [2805] := 46, [2806] := 48, [2807] := 48, [2808] := 48, [2809] := 48, [2810] := 48, [2811] := 48, [2812] := 48, [2813] := 48, [2814] := 13, [2815] := 10, [2816] := 51, [2817] := 53, [2818] := 56, [2819] := 56,
        [2820] := 56, [2821] := 44, [2822] := 48, [2823] := 46, [2824] := 48, [2825] := 57, [2826] := 50, [2827] := 57, [2828] := 54, [2829] := 49, [2830] := 50, [2831] := 51, [2832] := 44, [2833] := 50, [2834] := 46, [2835] := 48, [2836] := 48, [2837] := 48, [2838] := 48, [2839] := 48, [2840] := 48, [2841] := 48, [2842] := 48, [2843] := 44, [2844] := 53, [2845] := 46, [2846] := 48, [2847] := 48, [2848] := 48, [2849] := 48, [2850] := 48, [2851] := 48, [2852] := 48, [2853] := 48, [2854] := 44, [2855] := 54, [2856] := 46, [2857] := 48, [2858] := 48, [2859] := 48, [2860] := 48, [2861] := 48, [2862] := 48, [2863] := 48, [2864] := 48, [2865] := 44, [2866] := 55, [2867] := 46, [2868] := 48, [2869] := 48, [2870] := 48, [2871] := 48, [2872] := 48, [2873] := 48, [2874] := 48, [2875] := 48, [2876] := 44, [2877] := 56, [2878] := 46, [2879] := 48,
        [2880] := 48, [2881] := 48, [2882] := 48, [2883] := 48, [2884] := 48, [2885] := 48, [2886] := 48, [2887] := 44, [2888] := 57, [2889] := 46, [2890] := 48, [2891] := 48, [2892] := 48, [2893] := 48, [2894] := 48, [2895] := 48, [2896] := 48, [2897] := 48, [2898] := 44, [2899] := 49, [2900] := 48, [2901] := 46, [2902] := 48, [2903] := 48, [2904] := 48, [2905] := 48, [2906] := 48, [2907] := 48, [2908] := 48, [2909] := 44, [2910] := 49, [2911] := 49, [2912] := 46, [2913] := 48, [2914] := 48, [2915] := 48, [2916] := 48, [2917] := 48, [2918] := 48, [2919] := 48, [2920] := 44, [2921] := 49, [2922] := 50, [2923] := 46, [2924] := 48, [2925] := 48, [2926] := 48, [2927] := 48, [2928] := 48, [2929] := 48, [2930] := 48, [2931] := 44, [2932] := 49, [2933] := 46, [2934] := 48, [2935] := 48, [2936] := 48, [2937] := 48, [2938] := 48, [2939] := 48,
        [2940] := 48, [2941] := 48, [2942] := 13, [2943] := 10, [2944] := 51, [2945] := 53, [2946] := 56, [2947] := 56, [2948] := 56, [2949] := 44, [2950] := 48, [2951] := 46, [2952] := 48, [2953] := 57, [2954] := 50, [2955] := 57, [2956] := 55, [2957] := 50, [2958] := 56, [2959] := 48, [2960] := 44, [2961] := 50, [2962] := 46, [2963] := 48, [2964] := 48, [2965] := 48, [2966] := 48, [2967] := 48, [2968] := 48, [2969] := 48, [2970] := 48, [2971] := 44, [2972] := 53, [2973] := 46, [2974] := 48, [2975] := 48, [2976] := 48, [2977] := 48, [2978] := 48, [2979] := 48, [2980] := 48, [2981] := 48, [2982] := 44, [2983] := 54, [2984] := 46, [2985] := 48, [2986] := 48, [2987] := 48, [2988] := 48, [2989] := 48, [2990] := 48, [2991] := 48, [2992] := 48, [2993] := 44, [2994] := 55, [2995] := 46, [2996] := 48, [2997] := 48, [2998] := 48, [2999] := 48,
        [3000] := 48, [3001] := 48, [3002] := 48, [3003] := 48, [3004] := 44, [3005] := 56, [3006] := 46, [3007] := 48, [3008] := 48, [3009] := 48, [3010] := 48, [3011] := 48, [3012] := 48, [3013] := 48, [3014] := 48, [3015] := 44, [3016] := 57, [3017] := 46, [3018] := 48, [3019] := 48, [3020] := 48, [3021] := 48, [3022] := 48, [3023] := 48, [3024] := 48, [3025] := 48, [3026] := 44, [3027] := 49, [3028] := 48, [3029] := 46, [3030] := 48, [3031] := 48, [3032] := 48, [3033] := 48, [3034] := 48, [3035] := 48, [3036] := 48, [3037] := 44, [3038] := 49, [3039] := 49, [3040] := 46, [3041] := 48, [3042] := 48, [3043] := 48, [3044] := 48, [3045] := 48, [3046] := 48, [3047] := 48, [3048] := 44, [3049] := 49, [3050] := 50, [3051] := 46, [3052] := 48, [3053] := 48, [3054] := 48, [3055] := 48, [3056] := 48, [3057] := 48, [3058] := 48, [3059] := 44,
        [3060] := 49, [3061] := 46, [3062] := 48, [3063] := 48, [3064] := 48, [3065] := 48, [3066] := 48, [3067] := 48, [3068] := 48, [3069] := 48, [3070] := 13, [3071] := 10, [3072] := 51, [3073] := 53, [3074] := 56, [3075] := 56, [3076] := 56, [3077] := 44, [3078] := 48, [3079] := 46, [3080] := 48, [3081] := 57, [3082] := 50, [3083] := 57, [3084] := 56, [3085] := 52, [3086] := 51, [3087] := 56, [3088] := 44, [3089] := 50, [3090] := 46, [3091] := 48, [3092] := 48, [3093] := 48, [3094] := 48, [3095] := 48, [3096] := 48, [3097] := 48, [3098] := 48, [3099] := 44, [3100] := 53, [3101] := 46, [3102] := 48, [3103] := 48, [3104] := 48, [3105] := 48, [3106] := 48, [3107] := 48, [3108] := 48, [3109] := 48, [3110] := 44, [3111] := 54, [3112] := 46, [3113] := 48, [3114] := 48, [3115] := 48, [3116] := 48, [3117] := 48, [3118] := 48, [3119] := 48,
        [3120] := 48, [3121] := 44, [3122] := 55, [3123] := 46, [3124] := 48, [3125] := 48, [3126] := 48, [3127] := 48, [3128] := 48, [3129] := 48, [3130] := 48, [3131] := 48, [3132] := 44, [3133] := 56, [3134] := 46, [3135] := 48, [3136] := 48, [3137] := 48, [3138] := 48, [3139] := 48, [3140] := 48, [3141] := 48, [3142] := 48, [3143] := 44, [3144] := 57, [3145] := 46, [3146] := 48, [3147] := 48, [3148] := 48, [3149] := 48, [3150] := 48, [3151] := 48, [3152] := 48, [3153] := 48, [3154] := 44, [3155] := 49, [3156] := 48, [3157] := 46, [3158] := 48, [3159] := 48, [3160] := 48, [3161] := 48, [3162] := 48, [3163] := 48, [3164] := 48, [3165] := 44, [3166] := 49, [3167] := 49, [3168] := 46, [3169] := 48, [3170] := 48, [3171] := 48, [3172] := 48, [3173] := 48, [3174] := 48, [3175] := 48, [3176] := 44, [3177] := 49, [3178] := 50, [3179] := 46,
        [3180] := 48, [3181] := 48, [3182] := 48, [3183] := 48, [3184] := 48, [3185] := 48, [3186] := 48, [3187] := 44, [3188] := 49, [3189] := 46, [3190] := 48, [3191] := 48, [3192] := 48, [3193] := 48, [3194] := 48, [3195] := 48, [3196] := 48, [3197] := 48, [3198] := 13, [3199] := 10, [3200] := 51, [3201] := 53, [3202] := 56, [3203] := 56, [3204] := 56, [3205] := 44, [3206] := 48, [3207] := 46, [3208] := 48, [3209] := 57, [3210] := 50, [3211] := 57, [3212] := 57, [3213] := 53, [3214] := 57, [3215] := 53, [3216] := 44, [3217] := 50, [3218] := 46, [3219] := 48, [3220] := 48, [3221] := 48, [3222] := 48, [3223] := 48, [3224] := 48, [3225] := 48, [3226] := 48, [3227] := 44, [3228] := 53, [3229] := 46, [3230] := 48, [3231] := 48, [3232] := 48, [3233] := 48, [3234] := 48, [3235] := 48, [3236] := 48, [3237] := 48, [3238] := 44, [3239] := 54,
        [3240] := 46, [3241] := 48, [3242] := 48, [3243] := 48, [3244] := 48, [3245] := 48, [3246] := 48, [3247] := 48, [3248] := 48, [3249] := 44, [3250] := 55, [3251] := 46, [3252] := 48, [3253] := 48, [3254] := 48, [3255] := 48, [3256] := 48, [3257] := 48, [3258] := 48, [3259] := 48, [3260] := 44, [3261] := 56, [3262] := 46, [3263] := 48, [3264] := 48, [3265] := 48, [3266] := 48, [3267] := 48, [3268] := 48, [3269] := 48, [3270] := 48, [3271] := 44, [3272] := 57, [3273] := 46, [3274] := 48, [3275] := 48, [3276] := 48, [3277] := 48, [3278] := 48, [3279] := 48, [3280] := 48, [3281] := 48, [3282] := 44, [3283] := 49, [3284] := 48, [3285] := 46, [3286] := 48, [3287] := 48, [3288] := 48, [3289] := 48, [3290] := 48, [3291] := 48, [3292] := 48, [3293] := 44, [3294] := 49, [3295] := 49, [3296] := 46, [3297] := 48, [3298] := 48, [3299] := 48,
        [3300] := 48, [3301] := 48, [3302] := 48, [3303] := 48, [3304] := 44, [3305] := 49, [3306] := 50, [3307] := 46, [3308] := 48, [3309] := 48, [3310] := 48, [3311] := 48, [3312] := 48, [3313] := 48, [3314] := 48, [3315] := 44, [3316] := 49, [3317] := 46, [3318] := 48, [3319] := 48, [3320] := 48, [3321] := 48, [3322] := 48, [3323] := 48, [3324] := 48, [3325] := 48, [3326] := 13, [3327] := 10, [3328] := 51, [3329] := 53, [3330] := 56, [3331] := 56, [3332] := 56, [3333] := 44, [3334] := 48, [3335] := 46, [3336] := 48, [3337] := 57, [3338] := 51, [3339] := 48, [3340] := 48, [3341] := 55, [3342] := 53, [3343] := 50, [3344] := 44, [3345] := 50, [3346] := 46, [3347] := 48, [3348] := 48, [3349] := 48, [3350] := 48, [3351] := 48, [3352] := 48, [3353] := 48, [3354] := 48, [3355] := 44, [3356] := 53, [3357] := 46, [3358] := 48, [3359] := 48,
        [3360] := 48, [3361] := 48, [3362] := 48, [3363] := 48, [3364] := 48, [3365] := 48, [3366] := 44, [3367] := 54, [3368] := 46, [3369] := 48, [3370] := 48, [3371] := 48, [3372] := 48, [3373] := 48, [3374] := 48, [3375] := 48, [3376] := 48, [3377] := 44, [3378] := 55, [3379] := 46, [3380] := 48, [3381] := 48, [3382] := 48, [3383] := 48, [3384] := 48, [3385] := 48, [3386] := 48, [3387] := 48, [3388] := 44, [3389] := 56, [3390] := 46, [3391] := 48, [3392] := 48, [3393] := 48, [3394] := 48, [3395] := 48, [3396] := 48, [3397] := 48, [3398] := 48, [3399] := 44, [3400] := 57, [3401] := 46, [3402] := 48, [3403] := 48, [3404] := 48, [3405] := 48, [3406] := 48, [3407] := 48, [3408] := 48, [3409] := 48, [3410] := 44, [3411] := 49, [3412] := 48, [3413] := 46, [3414] := 48, [3415] := 48, [3416] := 48, [3417] := 48, [3418] := 48, [3419] := 48,
        [3420] := 48, [3421] := 44, [3422] := 49, [3423] := 49, [3424] := 46, [3425] := 48, [3426] := 48, [3427] := 48, [3428] := 48, [3429] := 48, [3430] := 48, [3431] := 48, [3432] := 44, [3433] := 49, [3434] := 50, [3435] := 46, [3436] := 48, [3437] := 48, [3438] := 48, [3439] := 48, [3440] := 48, [3441] := 48, [3442] := 48, [3443] := 44, [3444] := 49, [3445] := 46, [3446] := 48, [3447] := 48, [3448] := 48, [3449] := 48, [3450] := 48, [3451] := 48, [3452] := 48, [3453] := 48, [3454] := 13, [3455] := 10, [3456] := 51, [3457] := 53, [3458] := 56, [3459] := 56, [3460] := 56, [3461] := 44, [3462] := 48, [3463] := 46, [3464] := 48, [3465] := 57, [3466] := 51, [3467] := 48, [3468] := 49, [3469] := 57, [3470] := 49, [3471] := 48, [3472] := 44, [3473] := 50, [3474] := 46, [3475] := 48, [3476] := 48, [3477] := 48, [3478] := 48, [3479] := 48,
        [3480] := 48, [3481] := 48, [3482] := 48, [3483] := 44, [3484] := 53, [3485] := 46, [3486] := 48, [3487] := 48, [3488] := 48, [3489] := 48, [3490] := 48, [3491] := 48, [3492] := 48, [3493] := 48, [3494] := 44, [3495] := 54, [3496] := 46, [3497] := 48, [3498] := 48, [3499] := 48, [3500] := 48, [3501] := 48, [3502] := 48, [3503] := 48, [3504] := 48, [3505] := 44, [3506] := 55, [3507] := 46, [3508] := 48, [3509] := 48, [3510] := 48, [3511] := 48, [3512] := 48, [3513] := 48, [3514] := 48, [3515] := 48, [3516] := 44, [3517] := 56, [3518] := 46, [3519] := 48, [3520] := 48, [3521] := 48, [3522] := 48, [3523] := 48, [3524] := 48, [3525] := 48, [3526] := 48, [3527] := 44, [3528] := 57, [3529] := 46, [3530] := 48, [3531] := 48, [3532] := 48, [3533] := 48, [3534] := 48, [3535] := 48, [3536] := 48, [3537] := 48, [3538] := 44, [3539] := 49,
        [3540] := 48, [3541] := 46, [3542] := 48, [3543] := 48, [3544] := 48, [3545] := 48, [3546] := 48, [3547] := 48, [3548] := 48, [3549] := 44, [3550] := 49, [3551] := 49, [3552] := 46, [3553] := 48, [3554] := 48, [3555] := 48, [3556] := 48, [3557] := 48, [3558] := 48, [3559] := 48, [3560] := 44, [3561] := 49, [3562] := 50, [3563] := 46, [3564] := 48, [3565] := 48, [3566] := 48, [3567] := 48, [3568] := 48, [3569] := 48, [3570] := 48, [3571] := 44, [3572] := 49, [3573] := 46, [3574] := 48, [3575] := 48, [3576] := 48, [3577] := 48, [3578] := 48, [3579] := 48, [3580] := 48, [3581] := 48, [3582] := 13, [3583] := 10, [3584] := 51, [3585] := 53, [3586] := 56, [3587] := 56, [3588] := 56, [3589] := 44, [3590] := 48, [3591] := 46, [3592] := 48, [3593] := 57, [3594] := 51, [3595] := 48, [3596] := 51, [3597] := 48, [3598] := 54, [3599] := 55,
        [3600] := 44, [3601] := 50, [3602] := 46, [3603] := 48, [3604] := 48, [3605] := 48, [3606] := 48, [3607] := 48, [3608] := 48, [3609] := 48, [3610] := 48, [3611] := 44, [3612] := 53, [3613] := 46, [3614] := 48, [3615] := 48, [3616] := 48, [3617] := 48, [3618] := 48, [3619] := 48, [3620] := 48, [3621] := 48, [3622] := 44, [3623] := 54, [3624] := 46, [3625] := 48, [3626] := 48, [3627] := 48, [3628] := 48, [3629] := 48, [3630] := 48, [3631] := 48, [3632] := 48, [3633] := 44, [3634] := 55, [3635] := 46, [3636] := 48, [3637] := 48, [3638] := 48, [3639] := 48, [3640] := 48, [3641] := 48, [3642] := 48, [3643] := 48, [3644] := 44, [3645] := 56, [3646] := 46, [3647] := 48, [3648] := 48, [3649] := 48, [3650] := 48, [3651] := 48, [3652] := 48, [3653] := 48, [3654] := 48, [3655] := 44, [3656] := 57, [3657] := 46, [3658] := 48, [3659] := 48,
        [3660] := 48, [3661] := 48, [3662] := 48, [3663] := 48, [3664] := 48, [3665] := 48, [3666] := 44, [3667] := 49, [3668] := 48, [3669] := 46, [3670] := 48, [3671] := 48, [3672] := 48, [3673] := 48, [3674] := 48, [3675] := 48, [3676] := 48, [3677] := 44, [3678] := 49, [3679] := 49, [3680] := 46, [3681] := 48, [3682] := 48, [3683] := 48, [3684] := 48, [3685] := 48, [3686] := 48, [3687] := 48, [3688] := 44, [3689] := 49, [3690] := 50, [3691] := 46, [3692] := 48, [3693] := 48, [3694] := 48, [3695] := 48, [3696] := 48, [3697] := 48, [3698] := 48, [3699] := 44, [3700] := 49, [3701] := 46, [3702] := 48, [3703] := 48, [3704] := 48, [3705] := 48, [3706] := 48, [3707] := 48, [3708] := 48, [3709] := 48, [3710] := 13, [3711] := 10, [3712] := 51, [3713] := 53, [3714] := 56, [3715] := 56, [3716] := 56, [3717] := 44, [3718] := 48, [3719] := 46,
        [3720] := 48, [3721] := 57, [3722] := 51, [3723] := 48, [3724] := 52, [3725] := 50, [3726] := 50, [3727] := 53, [3728] := 44, [3729] := 50, [3730] := 46, [3731] := 48, [3732] := 48, [3733] := 48, [3734] := 48, [3735] := 48, [3736] := 48, [3737] := 48, [3738] := 48, [3739] := 44, [3740] := 53, [3741] := 46, [3742] := 48, [3743] := 48, [3744] := 48, [3745] := 48, [3746] := 48, [3747] := 48, [3748] := 48, [3749] := 48, [3750] := 44, [3751] := 54, [3752] := 46, [3753] := 48, [3754] := 48, [3755] := 48, [3756] := 48, [3757] := 48, [3758] := 48, [3759] := 48, [3760] := 48, [3761] := 44, [3762] := 55, [3763] := 46, [3764] := 48, [3765] := 48, [3766] := 48, [3767] := 48, [3768] := 48, [3769] := 48, [3770] := 48, [3771] := 48, [3772] := 44, [3773] := 56, [3774] := 46, [3775] := 48, [3776] := 48, [3777] := 48, [3778] := 48, [3779] := 48,
        [3780] := 48, [3781] := 48, [3782] := 48, [3783] := 44, [3784] := 57, [3785] := 46, [3786] := 48, [3787] := 48, [3788] := 48, [3789] := 48, [3790] := 48, [3791] := 48, [3792] := 48, [3793] := 48, [3794] := 44, [3795] := 49, [3796] := 48, [3797] := 46, [3798] := 48, [3799] := 48, [3800] := 48, [3801] := 48, [3802] := 48, [3803] := 48, [3804] := 48, [3805] := 44, [3806] := 49, [3807] := 49, [3808] := 46, [3809] := 48, [3810] := 48, [3811] := 48, [3812] := 48, [3813] := 48, [3814] := 48, [3815] := 48, [3816] := 44, [3817] := 49, [3818] := 50, [3819] := 46, [3820] := 48, [3821] := 48, [3822] := 48, [3823] := 48, [3824] := 48, [3825] := 48, [3826] := 48, [3827] := 44, [3828] := 49, [3829] := 46, [3830] := 48, [3831] := 48, [3832] := 48, [3833] := 48, [3834] := 48, [3835] := 48, [3836] := 48, [3837] := 48, [3838] := 13, [3839] := 10,
        [3840] := 51, [3841] := 53, [3842] := 56, [3843] := 56, [3844] := 56, [3845] := 44, [3846] := 48, [3847] := 46, [3848] := 48, [3849] := 57, [3850] := 51, [3851] := 48, [3852] := 53, [3853] := 51, [3854] := 56, [3855] := 50, [3856] := 44, [3857] := 50, [3858] := 46, [3859] := 48, [3860] := 48, [3861] := 48, [3862] := 48, [3863] := 48, [3864] := 48, [3865] := 48, [3866] := 48, [3867] := 44, [3868] := 53, [3869] := 46, [3870] := 48, [3871] := 48, [3872] := 48, [3873] := 48, [3874] := 48, [3875] := 48, [3876] := 48, [3877] := 48, [3878] := 44, [3879] := 54, [3880] := 46, [3881] := 48, [3882] := 48, [3883] := 48, [3884] := 48, [3885] := 48, [3886] := 48, [3887] := 48, [3888] := 48, [3889] := 44, [3890] := 55, [3891] := 46, [3892] := 48, [3893] := 48, [3894] := 48, [3895] := 48, [3896] := 48, [3897] := 48, [3898] := 48, [3899] := 48,
        [3900] := 44, [3901] := 56, [3902] := 46, [3903] := 48, [3904] := 48, [3905] := 48, [3906] := 48, [3907] := 48, [3908] := 48, [3909] := 48, [3910] := 48, [3911] := 44, [3912] := 57, [3913] := 46, [3914] := 48, [3915] := 48, [3916] := 48, [3917] := 48, [3918] := 48, [3919] := 48, [3920] := 48, [3921] := 48, [3922] := 44, [3923] := 49, [3924] := 48, [3925] := 46, [3926] := 48, [3927] := 48, [3928] := 48, [3929] := 48, [3930] := 48, [3931] := 48, [3932] := 48, [3933] := 44, [3934] := 49, [3935] := 49, [3936] := 46, [3937] := 48, [3938] := 48, [3939] := 48, [3940] := 48, [3941] := 48, [3942] := 48, [3943] := 48, [3944] := 44, [3945] := 49, [3946] := 50, [3947] := 46, [3948] := 48, [3949] := 48, [3950] := 48, [3951] := 48, [3952] := 48, [3953] := 48, [3954] := 48, [3955] := 44, [3956] := 49, [3957] := 46, [3958] := 48, [3959] := 48,
        [3960] := 48, [3961] := 48, [3962] := 48, [3963] := 48, [3964] := 48, [3965] := 48, [3966] := 13, [3967] := 10, [3968] := 51, [3969] := 53, [3970] := 56, [3971] := 56, [3972] := 56, [3973] := 44, [3974] := 48, [3975] := 46, [3976] := 48, [3977] := 57, [3978] := 51, [3979] := 48, [3980] := 54, [3981] := 53, [3982] := 52, [3983] := 48, [3984] := 44, [3985] := 50, [3986] := 46, [3987] := 48, [3988] := 48, [3989] := 48, [3990] := 48, [3991] := 48, [3992] := 48, [3993] := 48, [3994] := 48, [3995] := 44, [3996] := 53, [3997] := 46, [3998] := 48, [3999] := 48, [4000] := 48, [4001] := 48, [4002] := 48, [4003] := 48, [4004] := 48, [4005] := 48, [4006] := 44, [4007] := 54, [4008] := 46, [4009] := 48, [4010] := 48, [4011] := 48, [4012] := 48, [4013] := 48, [4014] := 48, [4015] := 48, [4016] := 48, [4017] := 44, [4018] := 55, [4019] := 46,
        [4020] := 48, [4021] := 48, [4022] := 48, [4023] := 48, [4024] := 48, [4025] := 48, [4026] := 48, [4027] := 48, [4028] := 44, [4029] := 56, [4030] := 46, [4031] := 48, [4032] := 48, [4033] := 48, [4034] := 48, [4035] := 48, [4036] := 48, [4037] := 48, [4038] := 48, [4039] := 44, [4040] := 57, [4041] := 46, [4042] := 48, [4043] := 48, [4044] := 48, [4045] := 48, [4046] := 48, [4047] := 48, [4048] := 48, [4049] := 48, [4050] := 44, [4051] := 49, [4052] := 48, [4053] := 46, [4054] := 48, [4055] := 48, [4056] := 48, [4057] := 48, [4058] := 48, [4059] := 48, [4060] := 48, [4061] := 44, [4062] := 49, [4063] := 49, [4064] := 46, [4065] := 48, [4066] := 48, [4067] := 48, [4068] := 48, [4069] := 48, [4070] := 48, [4071] := 48, [4072] := 44, [4073] := 49, [4074] := 50, [4075] := 46, [4076] := 48, [4077] := 48, [4078] := 48, [4079] := 48,
        [4080] := 48, [4081] := 48, [4082] := 48, [4083] := 44, [4084] := 49, [4085] := 46, [4086] := 48, [4087] := 48, [4088] := 48, [4089] := 48, [4090] := 48, [4091] := 48, [4092] := 48, [4093] := 48, [4094] := 13, [4095] := 10, [4096] := 51, [4097] := 53, [4098] := 56, [4099] := 56, [4100] := 56, [4101] := 44, [4102] := 48, [4103] := 46, [4104] := 48, [4105] := 57, [4106] := 51, [4107] := 48, [4108] := 55, [4109] := 54, [4110] := 57, [4111] := 55, [4112] := 44, [4113] := 50, [4114] := 46, [4115] := 48, [4116] := 48, [4117] := 48, [4118] := 48, [4119] := 48, [4120] := 48, [4121] := 48, [4122] := 48, [4123] := 44, [4124] := 53, [4125] := 46, [4126] := 48, [4127] := 48, [4128] := 48, [4129] := 48, [4130] := 48, [4131] := 48, [4132] := 48, [4133] := 48, [4134] := 44, [4135] := 54, [4136] := 46, [4137] := 48, [4138] := 48, [4139] := 48,
        [4140] := 48, [4141] := 48, [4142] := 48, [4143] := 48, [4144] := 48, [4145] := 44, [4146] := 55, [4147] := 46, [4148] := 48, [4149] := 48, [4150] := 48, [4151] := 48, [4152] := 48, [4153] := 48, [4154] := 48, [4155] := 48, [4156] := 44, [4157] := 56, [4158] := 46, [4159] := 48, [4160] := 48, [4161] := 48, [4162] := 48, [4163] := 48, [4164] := 48, [4165] := 48, [4166] := 48, [4167] := 44, [4168] := 57, [4169] := 46, [4170] := 48, [4171] := 48, [4172] := 48, [4173] := 48, [4174] := 48, [4175] := 48, [4176] := 48, [4177] := 48, [4178] := 44, [4179] := 49, [4180] := 48, [4181] := 46, [4182] := 48, [4183] := 48, [4184] := 48, [4185] := 48, [4186] := 48, [4187] := 48, [4188] := 48, [4189] := 44, [4190] := 49, [4191] := 49, [4192] := 46, [4193] := 48, [4194] := 48, [4195] := 48, [4196] := 48, [4197] := 48, [4198] := 48, [4199] := 48,
        [4200] := 44, [4201] := 49, [4202] := 50, [4203] := 46, [4204] := 48, [4205] := 48, [4206] := 48, [4207] := 48, [4208] := 48, [4209] := 48, [4210] := 48, [4211] := 44, [4212] := 49, [4213] := 46, [4214] := 48, [4215] := 48, [4216] := 48, [4217] := 48, [4218] := 48, [4219] := 48, [4220] := 48, [4221] := 48, [4222] := 13, [4223] := 10, [4224] := 51, [4225] := 53, [4226] := 56, [4227] := 56, [4228] := 56, [4229] := 44, [4230] := 48, [4231] := 46, [4232] := 48, [4233] := 57, [4234] := 51, [4235] := 48, [4236] := 56, [4237] := 56, [4238] := 53, [4239] := 52, [4240] := 44, [4241] := 50, [4242] := 46, [4243] := 48, [4244] := 48, [4245] := 48, [4246] := 48, [4247] := 48, [4248] := 48, [4249] := 48, [4250] := 48, [4251] := 44, [4252] := 53, [4253] := 46, [4254] := 48, [4255] := 48, [4256] := 48, [4257] := 48, [4258] := 48, [4259] := 48,
        [4260] := 48, [4261] := 48, [4262] := 44, [4263] := 54, [4264] := 46, [4265] := 48, [4266] := 48, [4267] := 48, [4268] := 48, [4269] := 48, [4270] := 48, [4271] := 48, [4272] := 48, [4273] := 44, [4274] := 55, [4275] := 46, [4276] := 48, [4277] := 48, [4278] := 48, [4279] := 48, [4280] := 48, [4281] := 48, [4282] := 48, [4283] := 48, [4284] := 44, [4285] := 56, [4286] := 46, [4287] := 48, [4288] := 48, [4289] := 48, [4290] := 48, [4291] := 48, [4292] := 48, [4293] := 48, [4294] := 48, [4295] := 44, [4296] := 57, [4297] := 46, [4298] := 48, [4299] := 48, [4300] := 48, [4301] := 48, [4302] := 48, [4303] := 48, [4304] := 48, [4305] := 48, [4306] := 44, [4307] := 49, [4308] := 48, [4309] := 46, [4310] := 48, [4311] := 48, [4312] := 48, [4313] := 48, [4314] := 48, [4315] := 48, [4316] := 48, [4317] := 44, [4318] := 49, [4319] := 49,
        [4320] := 46, [4321] := 48, [4322] := 48, [4323] := 48, [4324] := 48, [4325] := 48, [4326] := 48, [4327] := 48, [4328] := 44, [4329] := 49, [4330] := 50, [4331] := 46, [4332] := 48, [4333] := 48, [4334] := 48, [4335] := 48, [4336] := 48, [4337] := 48, [4338] := 48, [4339] := 44, [4340] := 49, [4341] := 46, [4342] := 48, [4343] := 48, [4344] := 48, [4345] := 48, [4346] := 48, [4347] := 48, [4348] := 48, [4349] := 48, [4350] := 13, [4351] := 10, [4352] := 51, [4353] := 53, [4354] := 56, [4355] := 56, [4356] := 56, [4357] := 44, [4358] := 48, [4359] := 46, [4360] := 48, [4361] := 57, [4362] := 51, [4363] := 49, [4364] := 48, [4365] := 48, [4366] := 49, [4367] := 50, [4368] := 44, [4369] := 50, [4370] := 46, [4371] := 48, [4372] := 48, [4373] := 48, [4374] := 48, [4375] := 48, [4376] := 48, [4377] := 48, [4378] := 48, [4379] := 44,
        [4380] := 53, [4381] := 46, [4382] := 48, [4383] := 48, [4384] := 48, [4385] := 48, [4386] := 48, [4387] := 48, [4388] := 48, [4389] := 48, [4390] := 44, [4391] := 54, [4392] := 46, [4393] := 48, [4394] := 48, [4395] := 48, [4396] := 48, [4397] := 48, [4398] := 48, [4399] := 48, [4400] := 48, [4401] := 44, [4402] := 55, [4403] := 46, [4404] := 48, [4405] := 48, [4406] := 48, [4407] := 48, [4408] := 48, [4409] := 48, [4410] := 48, [4411] := 48, [4412] := 44, [4413] := 56, [4414] := 46, [4415] := 48, [4416] := 48, [4417] := 48, [4418] := 48, [4419] := 48, [4420] := 48, [4421] := 48, [4422] := 48, [4423] := 44, [4424] := 57, [4425] := 46, [4426] := 48, [4427] := 48, [4428] := 48, [4429] := 48, [4430] := 48, [4431] := 48, [4432] := 48, [4433] := 48, [4434] := 44, [4435] := 49, [4436] := 48, [4437] := 46, [4438] := 48, [4439] := 48,
        [4440] := 48, [4441] := 48, [4442] := 48, [4443] := 48, [4444] := 48, [4445] := 44, [4446] := 49, [4447] := 49, [4448] := 46, [4449] := 48, [4450] := 48, [4451] := 48, [4452] := 48, [4453] := 48, [4454] := 48, [4455] := 48, [4456] := 44, [4457] := 49, [4458] := 50, [4459] := 46, [4460] := 48, [4461] := 48, [4462] := 48, [4463] := 48, [4464] := 48, [4465] := 48, [4466] := 48, [4467] := 44, [4468] := 49, [4469] := 46, [4470] := 48, [4471] := 48, [4472] := 48, [4473] := 48, [4474] := 48, [4475] := 48, [4476] := 48, [4477] := 48, [4478] := 13, [4479] := 10, [4480] := 51, [4481] := 53, [4482] := 56, [4483] := 56, [4484] := 56, [4485] := 44, [4486] := 48, [4487] := 46, [4488] := 48, [4489] := 57, [4490] := 51, [4491] := 49, [4492] := 49, [4493] := 49, [4494] := 54, [4495] := 57, [4496] := 44, [4497] := 50, [4498] := 46, [4499] := 48,
        [4500] := 48, [4501] := 48, [4502] := 48, [4503] := 48, [4504] := 48, [4505] := 48, [4506] := 48, [4507] := 44, [4508] := 53, [4509] := 46, [4510] := 48, [4511] := 48, [4512] := 48, [4513] := 48, [4514] := 48, [4515] := 48, [4516] := 48, [4517] := 48, [4518] := 44, [4519] := 54, [4520] := 46, [4521] := 48, [4522] := 48, [4523] := 48, [4524] := 48, [4525] := 48, [4526] := 48, [4527] := 48, [4528] := 48, [4529] := 44, [4530] := 55, [4531] := 46, [4532] := 48, [4533] := 48, [4534] := 48, [4535] := 48, [4536] := 48, [4537] := 48, [4538] := 48, [4539] := 48, [4540] := 44, [4541] := 56, [4542] := 46, [4543] := 48, [4544] := 48, [4545] := 48, [4546] := 48, [4547] := 48, [4548] := 48, [4549] := 48, [4550] := 48, [4551] := 44, [4552] := 57, [4553] := 46, [4554] := 48, [4555] := 48, [4556] := 48, [4557] := 48, [4558] := 48, [4559] := 48,
        [4560] := 48, [4561] := 48, [4562] := 44, [4563] := 49, [4564] := 48, [4565] := 46, [4566] := 48, [4567] := 48, [4568] := 48, [4569] := 48, [4570] := 48, [4571] := 48, [4572] := 48, [4573] := 44, [4574] := 49, [4575] := 49, [4576] := 46, [4577] := 48, [4578] := 48, [4579] := 48, [4580] := 48, [4581] := 48, [4582] := 48, [4583] := 48, [4584] := 44, [4585] := 49, [4586] := 50, [4587] := 46, [4588] := 48, [4589] := 48, [4590] := 48, [4591] := 48, [4592] := 48, [4593] := 48, [4594] := 48, [4595] := 44, [4596] := 49, [4597] := 46, [4598] := 48, [4599] := 48, [4600] := 48, [4601] := 48, [4602] := 48, [4603] := 48, [4604] := 48, [4605] := 48, [4606] := 13, [4607] := 10, [4608] := 51, [4609] := 53, [4610] := 56, [4611] := 56, [4612] := 56, [4613] := 44, [4614] := 48, [4615] := 46, [4616] := 48, [4617] := 57, [4618] := 51, [4619] := 49,
        [4620] := 50, [4621] := 51, [4622] := 50, [4623] := 55, [4624] := 44, [4625] := 50, [4626] := 46, [4627] := 48, [4628] := 48, [4629] := 48, [4630] := 48, [4631] := 48, [4632] := 48, [4633] := 48, [4634] := 48, [4635] := 44, [4636] := 53, [4637] := 46, [4638] := 48, [4639] := 48, [4640] := 48, [4641] := 48, [4642] := 48, [4643] := 48, [4644] := 48, [4645] := 48, [4646] := 44, [4647] := 54, [4648] := 46, [4649] := 48, [4650] := 48, [4651] := 48, [4652] := 48, [4653] := 48, [4654] := 48, [4655] := 48, [4656] := 48, [4657] := 44, [4658] := 55, [4659] := 46, [4660] := 48, [4661] := 48, [4662] := 48, [4663] := 48, [4664] := 48, [4665] := 48, [4666] := 48, [4667] := 48, [4668] := 44, [4669] := 56, [4670] := 46, [4671] := 48, [4672] := 48, [4673] := 48, [4674] := 48, [4675] := 48, [4676] := 48, [4677] := 48, [4678] := 48, [4679] := 44,
        [4680] := 57, [4681] := 46, [4682] := 48, [4683] := 48, [4684] := 48, [4685] := 48, [4686] := 48, [4687] := 48, [4688] := 48, [4689] := 48, [4690] := 44, [4691] := 49, [4692] := 48, [4693] := 46, [4694] := 48, [4695] := 48, [4696] := 48, [4697] := 48, [4698] := 48, [4699] := 48, [4700] := 48, [4701] := 44, [4702] := 49, [4703] := 49, [4704] := 46, [4705] := 48, [4706] := 48, [4707] := 48, [4708] := 48, [4709] := 48, [4710] := 48, [4711] := 48, [4712] := 44, [4713] := 49, [4714] := 50, [4715] := 46, [4716] := 48, [4717] := 48, [4718] := 48, [4719] := 48, [4720] := 48, [4721] := 48, [4722] := 48, [4723] := 44, [4724] := 49, [4725] := 46, [4726] := 48, [4727] := 48, [4728] := 48, [4729] := 48, [4730] := 48, [4731] := 48, [4732] := 48, [4733] := 48, [4734] := 13, [4735] := 10, [4736] := 51, [4737] := 53, [4738] := 56, [4739] := 56,
        [4740] := 56, [4741] := 44, [4742] := 48, [4743] := 46, [4744] := 48, [4745] := 57, [4746] := 51, [4747] := 49, [4748] := 51, [4749] := 52, [4750] := 56, [4751] := 52, [4752] := 44, [4753] := 50, [4754] := 46, [4755] := 48, [4756] := 48, [4757] := 48, [4758] := 48, [4759] := 48, [4760] := 48, [4761] := 48, [4762] := 48, [4763] := 44, [4764] := 53, [4765] := 46, [4766] := 48, [4767] := 48, [4768] := 48, [4769] := 48, [4770] := 48, [4771] := 48, [4772] := 48, [4773] := 48, [4774] := 44, [4775] := 54, [4776] := 46, [4777] := 48, [4778] := 48, [4779] := 48, [4780] := 48, [4781] := 48, [4782] := 48, [4783] := 48, [4784] := 48, [4785] := 44, [4786] := 55, [4787] := 46, [4788] := 48, [4789] := 48, [4790] := 48, [4791] := 48, [4792] := 48, [4793] := 48, [4794] := 48, [4795] := 48, [4796] := 44, [4797] := 56, [4798] := 46, [4799] := 48,
        [4800] := 48, [4801] := 48, [4802] := 48, [4803] := 48, [4804] := 48, [4805] := 48, [4806] := 48, [4807] := 44, [4808] := 57, [4809] := 46, [4810] := 48, [4811] := 48, [4812] := 48, [4813] := 48, [4814] := 48, [4815] := 48, [4816] := 48, [4817] := 48, [4818] := 44, [4819] := 49, [4820] := 48, [4821] := 46, [4822] := 48, [4823] := 48, [4824] := 48, [4825] := 48, [4826] := 48, [4827] := 48, [4828] := 48, [4829] := 44, [4830] := 49, [4831] := 49, [4832] := 46, [4833] := 48, [4834] := 48, [4835] := 48, [4836] := 48, [4837] := 48, [4838] := 48, [4839] := 48, [4840] := 44, [4841] := 49, [4842] := 50, [4843] := 46, [4844] := 48, [4845] := 48, [4846] := 48, [4847] := 48, [4848] := 48, [4849] := 48, [4850] := 48, [4851] := 44, [4852] := 49, [4853] := 46, [4854] := 48, [4855] := 48, [4856] := 48, [4857] := 48, [4858] := 48, [4859] := 48,
        [4860] := 48, [4861] := 48, [4862] := 13, [4863] := 10, [4864] := 51, [4865] := 53, [4866] := 56, [4867] := 56, [4868] := 56, [4869] := 44, [4870] := 48, [4871] := 46, [4872] := 48, [4873] := 57, [4874] := 51, [4875] := 49, [4876] := 52, [4877] := 54, [4878] := 52, [4879] := 49, [4880] := 44, [4881] := 50, [4882] := 46, [4883] := 48, [4884] := 48, [4885] := 48, [4886] := 48, [4887] := 48, [4888] := 48, [4889] := 48, [4890] := 48, [4891] := 44, [4892] := 53, [4893] := 46, [4894] := 48, [4895] := 48, [4896] := 48, [4897] := 48, [4898] := 48, [4899] := 48, [4900] := 48, [4901] := 48, [4902] := 44, [4903] := 54, [4904] := 46, [4905] := 48, [4906] := 48, [4907] := 48, [4908] := 48, [4909] := 48, [4910] := 48, [4911] := 48, [4912] := 48, [4913] := 44, [4914] := 55, [4915] := 46, [4916] := 48, [4917] := 48, [4918] := 48, [4919] := 48,
        [4920] := 48, [4921] := 48, [4922] := 48, [4923] := 48, [4924] := 44, [4925] := 56, [4926] := 46, [4927] := 48, [4928] := 48, [4929] := 48, [4930] := 48, [4931] := 48, [4932] := 48, [4933] := 48, [4934] := 48, [4935] := 44, [4936] := 57, [4937] := 46, [4938] := 48, [4939] := 48, [4940] := 48, [4941] := 48, [4942] := 48, [4943] := 48, [4944] := 48, [4945] := 48, [4946] := 44, [4947] := 49, [4948] := 48, [4949] := 46, [4950] := 48, [4951] := 48, [4952] := 48, [4953] := 48, [4954] := 48, [4955] := 48, [4956] := 48, [4957] := 44, [4958] := 49, [4959] := 49, [4960] := 46, [4961] := 48, [4962] := 48, [4963] := 48, [4964] := 48, [4965] := 48, [4966] := 48, [4967] := 48, [4968] := 44, [4969] := 49, [4970] := 50, [4971] := 46, [4972] := 48, [4973] := 48, [4974] := 48, [4975] := 48, [4976] := 48, [4977] := 48, [4978] := 48, [4979] := 44,
        [4980] := 49, [4981] := 46, [4982] := 48, [4983] := 48, [4984] := 48, [4985] := 48, [4986] := 48, [4987] := 48, [4988] := 48, [4989] := 48, [4990] := 13, [4991] := 10, [4992] := 51, [4993] := 53, [4994] := 56, [4995] := 56, [4996] := 56, [4997] := 44, [4998] := 48, [4999] := 46, [5000] := 48, [5001] := 57, [5002] := 51, [5003] := 49, [5004] := 53, [5005] := 55, [5006] := 57, [5007] := 56, [5008] := 44, [5009] := 50, [5010] := 46, [5011] := 48, [5012] := 48, [5013] := 48, [5014] := 48, [5015] := 48, [5016] := 48, [5017] := 48, [5018] := 48, [5019] := 44, [5020] := 53, [5021] := 46, [5022] := 48, [5023] := 48, [5024] := 48, [5025] := 48, [5026] := 48, [5027] := 48, [5028] := 48, [5029] := 48, [5030] := 44, [5031] := 54, [5032] := 46, [5033] := 48, [5034] := 48, [5035] := 48, [5036] := 48, [5037] := 48, [5038] := 48, [5039] := 48,
        [5040] := 48, [5041] := 44, [5042] := 55, [5043] := 46, [5044] := 48, [5045] := 48, [5046] := 48, [5047] := 48, [5048] := 48, [5049] := 48, [5050] := 48, [5051] := 48, [5052] := 44, [5053] := 56, [5054] := 46, [5055] := 48, [5056] := 48, [5057] := 48, [5058] := 48, [5059] := 48, [5060] := 48, [5061] := 48, [5062] := 48, [5063] := 44, [5064] := 57, [5065] := 46, [5066] := 48, [5067] := 48, [5068] := 48, [5069] := 48, [5070] := 48, [5071] := 48, [5072] := 48, [5073] := 48, [5074] := 44, [5075] := 49, [5076] := 48, [5077] := 46, [5078] := 48, [5079] := 48, [5080] := 48, [5081] := 48, [5082] := 48, [5083] := 48, [5084] := 48, [5085] := 44, [5086] := 49, [5087] := 49, [5088] := 46, [5089] := 48, [5090] := 48, [5091] := 48, [5092] := 48, [5093] := 48, [5094] := 48, [5095] := 48, [5096] := 44, [5097] := 49, [5098] := 50, [5099] := 46,
        [5100] := 48, [5101] := 48, [5102] := 48, [5103] := 48, [5104] := 48, [5105] := 48, [5106] := 48, [5107] := 44, [5108] := 49, [5109] := 46, [5110] := 48, [5111] := 48, [5112] := 48, [5113] := 48, [5114] := 48, [5115] := 48, [5116] := 48, [5117] := 48, [5118] := 13, [5119] := 10, [5120] := 51, [5121] := 53, [5122] := 56, [5123] := 56, [5124] := 56, [5125] := 44, [5126] := 48, [5127] := 46, [5128] := 48, [5129] := 57, [5130] := 51, [5131] := 49, [5132] := 54, [5133] := 57, [5134] := 53, [5135] := 54, [5136] := 44, [5137] := 50, [5138] := 46, [5139] := 48, [5140] := 48, [5141] := 48, [5142] := 48, [5143] := 48, [5144] := 48, [5145] := 48, [5146] := 48, [5147] := 44, [5148] := 53, [5149] := 46, [5150] := 48, [5151] := 48, [5152] := 48, [5153] := 48, [5154] := 48, [5155] := 48, [5156] := 48, [5157] := 48, [5158] := 44, [5159] := 54,
        [5160] := 46, [5161] := 48, [5162] := 48, [5163] := 48, [5164] := 48, [5165] := 48, [5166] := 48, [5167] := 48, [5168] := 48, [5169] := 44, [5170] := 55, [5171] := 46, [5172] := 48, [5173] := 48, [5174] := 48, [5175] := 48, [5176] := 48, [5177] := 48, [5178] := 48, [5179] := 48, [5180] := 44, [5181] := 56, [5182] := 46, [5183] := 48, [5184] := 48, [5185] := 48, [5186] := 48, [5187] := 48, [5188] := 48, [5189] := 48, [5190] := 48, [5191] := 44, [5192] := 57, [5193] := 46, [5194] := 48, [5195] := 48, [5196] := 48, [5197] := 48, [5198] := 48, [5199] := 48, [5200] := 48, [5201] := 48, [5202] := 44, [5203] := 49, [5204] := 48, [5205] := 46, [5206] := 48, [5207] := 48, [5208] := 48, [5209] := 48, [5210] := 48, [5211] := 48, [5212] := 48, [5213] := 44, [5214] := 49, [5215] := 49, [5216] := 46, [5217] := 48, [5218] := 48, [5219] := 48,
        [5220] := 48, [5221] := 48, [5222] := 48, [5223] := 48, [5224] := 44, [5225] := 49, [5226] := 50, [5227] := 46, [5228] := 48, [5229] := 48, [5230] := 48, [5231] := 48, [5232] := 48, [5233] := 48, [5234] := 48, [5235] := 44, [5236] := 49, [5237] := 46, [5238] := 48, [5239] := 48, [5240] := 48, [5241] := 48, [5242] := 48, [5243] := 48, [5244] := 48, [5245] := 48, [5246] := 13, [5247] := 10, [5248] := 51, [5249] := 53, [5250] := 56, [5251] := 56, [5252] := 56, [5253] := 44, [5254] := 48, [5255] := 46, [5256] := 48, [5257] := 57, [5258] := 51, [5259] := 49, [5260] := 56, [5261] := 49, [5262] := 49, [5263] := 52, [5264] := 44, [5265] := 50, [5266] := 46, [5267] := 48, [5268] := 48, [5269] := 48, [5270] := 48, [5271] := 48, [5272] := 48, [5273] := 48, [5274] := 48, [5275] := 44, [5276] := 53, [5277] := 46, [5278] := 48, [5279] := 48,
        [5280] := 48, [5281] := 48, [5282] := 48, [5283] := 48, [5284] := 48, [5285] := 48, [5286] := 44, [5287] := 54, [5288] := 46, [5289] := 48, [5290] := 48, [5291] := 48, [5292] := 48, [5293] := 48, [5294] := 48, [5295] := 48, [5296] := 48, [5297] := 44, [5298] := 55, [5299] := 46, [5300] := 48, [5301] := 48, [5302] := 48, [5303] := 48, [5304] := 48, [5305] := 48, [5306] := 48, [5307] := 48, [5308] := 44, [5309] := 56, [5310] := 46, [5311] := 48, [5312] := 48, [5313] := 48, [5314] := 48, [5315] := 48, [5316] := 48, [5317] := 48, [5318] := 48, [5319] := 44, [5320] := 57, [5321] := 46, [5322] := 48, [5323] := 48, [5324] := 48, [5325] := 48, [5326] := 48, [5327] := 48, [5328] := 48, [5329] := 48, [5330] := 44, [5331] := 49, [5332] := 48, [5333] := 46, [5334] := 48, [5335] := 48, [5336] := 48, [5337] := 48, [5338] := 48, [5339] := 48,
        [5340] := 48, [5341] := 44, [5342] := 49, [5343] := 49, [5344] := 46, [5345] := 48, [5346] := 48, [5347] := 48, [5348] := 48, [5349] := 48, [5350] := 48, [5351] := 48, [5352] := 44, [5353] := 49, [5354] := 50, [5355] := 46, [5356] := 48, [5357] := 48, [5358] := 48, [5359] := 48, [5360] := 48, [5361] := 48, [5362] := 48, [5363] := 44, [5364] := 49, [5365] := 46, [5366] := 48, [5367] := 48, [5368] := 48, [5369] := 48, [5370] := 48, [5371] := 48, [5372] := 48, [5373] := 48, [5374] := 13, [5375] := 10, [5376] := 51, [5377] := 53, [5378] := 56, [5379] := 56, [5380] := 56, [5381] := 44, [5382] := 48, [5383] := 46, [5384] := 48, [5385] := 57, [5386] := 51, [5387] := 49, [5388] := 57, [5389] := 50, [5390] := 55, [5391] := 49, [5392] := 44, [5393] := 50, [5394] := 46, [5395] := 48, [5396] := 48, [5397] := 48, [5398] := 48, [5399] := 48,
        [5400] := 48, [5401] := 48, [5402] := 48, [5403] := 44, [5404] := 53, [5405] := 46, [5406] := 48, [5407] := 48, [5408] := 48, [5409] := 48, [5410] := 48, [5411] := 48, [5412] := 48, [5413] := 48, [5414] := 44, [5415] := 54, [5416] := 46, [5417] := 48, [5418] := 48, [5419] := 48, [5420] := 48, [5421] := 48, [5422] := 48, [5423] := 48, [5424] := 48, [5425] := 44, [5426] := 55, [5427] := 46, [5428] := 48, [5429] := 48, [5430] := 48, [5431] := 48, [5432] := 48, [5433] := 48, [5434] := 48, [5435] := 48, [5436] := 44, [5437] := 56, [5438] := 46, [5439] := 48, [5440] := 48, [5441] := 48, [5442] := 48, [5443] := 48, [5444] := 48, [5445] := 48, [5446] := 48, [5447] := 44, [5448] := 57, [5449] := 46, [5450] := 48, [5451] := 48, [5452] := 48, [5453] := 48, [5454] := 48, [5455] := 48, [5456] := 48, [5457] := 48, [5458] := 44, [5459] := 49,
        [5460] := 48, [5461] := 46, [5462] := 48, [5463] := 48, [5464] := 48, [5465] := 48, [5466] := 48, [5467] := 48, [5468] := 48, [5469] := 44, [5470] := 49, [5471] := 49, [5472] := 46, [5473] := 48, [5474] := 48, [5475] := 48, [5476] := 48, [5477] := 48, [5478] := 48, [5479] := 48, [5480] := 44, [5481] := 49, [5482] := 50, [5483] := 46, [5484] := 48, [5485] := 48, [5486] := 48, [5487] := 48, [5488] := 48, [5489] := 48, [5490] := 48, [5491] := 44, [5492] := 49, [5493] := 46, [5494] := 48, [5495] := 48, [5496] := 48, [5497] := 48, [5498] := 48, [5499] := 48, [5500] := 48, [5501] := 48, [5502] := 13, [5503] := 10, [5504] := 51, [5505] := 53, [5506] := 56, [5507] := 56, [5508] := 56, [5509] := 44, [5510] := 48, [5511] := 46, [5512] := 48, [5513] := 57, [5514] := 51, [5515] := 50, [5516] := 48, [5517] := 52, [5518] := 50, [5519] := 56,
        [5520] := 44, [5521] := 50, [5522] := 46, [5523] := 48, [5524] := 48, [5525] := 48, [5526] := 48, [5527] := 48, [5528] := 48, [5529] := 48, [5530] := 48, [5531] := 44, [5532] := 53, [5533] := 46, [5534] := 48, [5535] := 48, [5536] := 48, [5537] := 48, [5538] := 48, [5539] := 48, [5540] := 48, [5541] := 48, [5542] := 44, [5543] := 54, [5544] := 46, [5545] := 48, [5546] := 48, [5547] := 48, [5548] := 48, [5549] := 48, [5550] := 48, [5551] := 48, [5552] := 48, [5553] := 44, [5554] := 55, [5555] := 46, [5556] := 48, [5557] := 48, [5558] := 48, [5559] := 48, [5560] := 48, [5561] := 48, [5562] := 48, [5563] := 48, [5564] := 44, [5565] := 56, [5566] := 46, [5567] := 48, [5568] := 48, [5569] := 48, [5570] := 48, [5571] := 48, [5572] := 48, [5573] := 48, [5574] := 48, [5575] := 44, [5576] := 57, [5577] := 46, [5578] := 48, [5579] := 48,
        [5580] := 48, [5581] := 48, [5582] := 48, [5583] := 48, [5584] := 48, [5585] := 48, [5586] := 44, [5587] := 49, [5588] := 48, [5589] := 46, [5590] := 48, [5591] := 48, [5592] := 48, [5593] := 48, [5594] := 48, [5595] := 48, [5596] := 48, [5597] := 44, [5598] := 49, [5599] := 49, [5600] := 46, [5601] := 48, [5602] := 48, [5603] := 48, [5604] := 48, [5605] := 48, [5606] := 48, [5607] := 48, [5608] := 44, [5609] := 49, [5610] := 50, [5611] := 46, [5612] := 48, [5613] := 48, [5614] := 48, [5615] := 48, [5616] := 48, [5617] := 48, [5618] := 48, [5619] := 44, [5620] := 49, [5621] := 46, [5622] := 48, [5623] := 48, [5624] := 48, [5625] := 48, [5626] := 48, [5627] := 48, [5628] := 48, [5629] := 48, [5630] := 13, [5631] := 10, [5632] := 51, [5633] := 53, [5634] := 56, [5635] := 56, [5636] := 56, [5637] := 44, [5638] := 48, [5639] := 46,
        [5640] := 48, [5641] := 57, [5642] := 51, [5643] := 50, [5644] := 49, [5645] := 53, [5646] := 56, [5647] := 53, [5648] := 44, [5649] := 50, [5650] := 46, [5651] := 48, [5652] := 48, [5653] := 48, [5654] := 48, [5655] := 48, [5656] := 48, [5657] := 48, [5658] := 48, [5659] := 44, [5660] := 53, [5661] := 46, [5662] := 48, [5663] := 48, [5664] := 48, [5665] := 48, [5666] := 48, [5667] := 48, [5668] := 48, [5669] := 48, [5670] := 44, [5671] := 54, [5672] := 46, [5673] := 48, [5674] := 48, [5675] := 48, [5676] := 48, [5677] := 48, [5678] := 48, [5679] := 48, [5680] := 48, [5681] := 44, [5682] := 55, [5683] := 46, [5684] := 48, [5685] := 48, [5686] := 48, [5687] := 48, [5688] := 48, [5689] := 48, [5690] := 48, [5691] := 48, [5692] := 44, [5693] := 56, [5694] := 46, [5695] := 48, [5696] := 48, [5697] := 48, [5698] := 48, [5699] := 48,
        [5700] := 48, [5701] := 48, [5702] := 48, [5703] := 44, [5704] := 57, [5705] := 46, [5706] := 48, [5707] := 48, [5708] := 48, [5709] := 48, [5710] := 48, [5711] := 48, [5712] := 48, [5713] := 48, [5714] := 44, [5715] := 49, [5716] := 48, [5717] := 46, [5718] := 48, [5719] := 48, [5720] := 48, [5721] := 48, [5722] := 48, [5723] := 48, [5724] := 48, [5725] := 44, [5726] := 49, [5727] := 49, [5728] := 46, [5729] := 48, [5730] := 48, [5731] := 48, [5732] := 48, [5733] := 48, [5734] := 48, [5735] := 48, [5736] := 44, [5737] := 49, [5738] := 50, [5739] := 46, [5740] := 48, [5741] := 48, [5742] := 48, [5743] := 48, [5744] := 48, [5745] := 48, [5746] := 48, [5747] := 44, [5748] := 49, [5749] := 46, [5750] := 48, [5751] := 48, [5752] := 48, [5753] := 48, [5754] := 48, [5755] := 48, [5756] := 48, [5757] := 48, [5758] := 13, [5759] := 10,
        [5760] := 51, [5761] := 53, [5762] := 56, [5763] := 56, [5764] := 56, [5765] := 44, [5766] := 48, [5767] := 46, [5768] := 48, [5769] := 57, [5770] := 51, [5771] := 50, [5772] := 50, [5773] := 55, [5774] := 52, [5775] := 52, [5776] := 44, [5777] := 50, [5778] := 46, [5779] := 48, [5780] := 48, [5781] := 48, [5782] := 48, [5783] := 48, [5784] := 48, [5785] := 48, [5786] := 48, [5787] := 44, [5788] := 53, [5789] := 46, [5790] := 48, [5791] := 48, [5792] := 48, [5793] := 48, [5794] := 48, [5795] := 48, [5796] := 48, [5797] := 48, [5798] := 44, [5799] := 54, [5800] := 46, [5801] := 48, [5802] := 48, [5803] := 48, [5804] := 48, [5805] := 48, [5806] := 48, [5807] := 48, [5808] := 48, [5809] := 44, [5810] := 55, [5811] := 46, [5812] := 48, [5813] := 48, [5814] := 48, [5815] := 48, [5816] := 48, [5817] := 48, [5818] := 48, [5819] := 48,
        [5820] := 44, [5821] := 56, [5822] := 46, [5823] := 48, [5824] := 48, [5825] := 48, [5826] := 48, [5827] := 48, [5828] := 48, [5829] := 48, [5830] := 48, [5831] := 44, [5832] := 57, [5833] := 46, [5834] := 48, [5835] := 48, [5836] := 48, [5837] := 48, [5838] := 48, [5839] := 48, [5840] := 48, [5841] := 48, [5842] := 44, [5843] := 49, [5844] := 48, [5845] := 46, [5846] := 48, [5847] := 48, [5848] := 48, [5849] := 48, [5850] := 48, [5851] := 48, [5852] := 48, [5853] := 44, [5854] := 49, [5855] := 49, [5856] := 46, [5857] := 48, [5858] := 48, [5859] := 48, [5860] := 48, [5861] := 48, [5862] := 48, [5863] := 48, [5864] := 44, [5865] := 49, [5866] := 50, [5867] := 46, [5868] := 48, [5869] := 48, [5870] := 48, [5871] := 48, [5872] := 48, [5873] := 48, [5874] := 48, [5875] := 44, [5876] := 49, [5877] := 46, [5878] := 48, [5879] := 48,
        [5880] := 48, [5881] := 48, [5882] := 48, [5883] := 48, [5884] := 48, [5885] := 48, [5886] := 13, [5887] := 10, [5888] := 51, [5889] := 53, [5890] := 56, [5891] := 56, [5892] := 56, [5893] := 44, [5894] := 48, [5895] := 46, [5896] := 48, [5897] := 57, [5898] := 51, [5899] := 50, [5900] := 51, [5901] := 57, [5902] := 48, [5903] := 49, [5904] := 44, [5905] := 50, [5906] := 46, [5907] := 48, [5908] := 48, [5909] := 48, [5910] := 48, [5911] := 48, [5912] := 48, [5913] := 48, [5914] := 48, [5915] := 44, [5916] := 53, [5917] := 46, [5918] := 48, [5919] := 48, [5920] := 48, [5921] := 48, [5922] := 48, [5923] := 48, [5924] := 48, [5925] := 48, [5926] := 44, [5927] := 54, [5928] := 46, [5929] := 48, [5930] := 48, [5931] := 48, [5932] := 48, [5933] := 48, [5934] := 48, [5935] := 48, [5936] := 48, [5937] := 44, [5938] := 55, [5939] := 46,
        [5940] := 48, [5941] := 48, [5942] := 48, [5943] := 48, [5944] := 48, [5945] := 48, [5946] := 48, [5947] := 48, [5948] := 44, [5949] := 56, [5950] := 46, [5951] := 48, [5952] := 48, [5953] := 48, [5954] := 48, [5955] := 48, [5956] := 48, [5957] := 48, [5958] := 48, [5959] := 44, [5960] := 57, [5961] := 46, [5962] := 48, [5963] := 48, [5964] := 48, [5965] := 48, [5966] := 48, [5967] := 48, [5968] := 48, [5969] := 48, [5970] := 44, [5971] := 49, [5972] := 48, [5973] := 46, [5974] := 48, [5975] := 48, [5976] := 48, [5977] := 48, [5978] := 48, [5979] := 48, [5980] := 48, [5981] := 44, [5982] := 49, [5983] := 49, [5984] := 46, [5985] := 48, [5986] := 48, [5987] := 48, [5988] := 48, [5989] := 48, [5990] := 48, [5991] := 48, [5992] := 44, [5993] := 49, [5994] := 50, [5995] := 46, [5996] := 48, [5997] := 48, [5998] := 48, [5999] := 48,
        [6000] := 48, [6001] := 48, [6002] := 48, [6003] := 44, [6004] := 49, [6005] := 46, [6006] := 48, [6007] := 48, [6008] := 48, [6009] := 48, [6010] := 48, [6011] := 48, [6012] := 48, [6013] := 48, [6014] := 13, [6015] := 10, [6016] := 51, [6017] := 53, [6018] := 56, [6019] := 56, [6020] := 56, [6021] := 44, [6022] := 48, [6023] := 46, [6024] := 48, [6025] := 57, [6026] := 51, [6027] := 50, [6028] := 53, [6029] := 48, [6030] := 53, [6031] := 57, [6032] := 44, [6033] := 50, [6034] := 46, [6035] := 48, [6036] := 48, [6037] := 48, [6038] := 48, [6039] := 48, [6040] := 48, [6041] := 48, [6042] := 48, [6043] := 44, [6044] := 53, [6045] := 46, [6046] := 48, [6047] := 48, [6048] := 48, [6049] := 48, [6050] := 48, [6051] := 48, [6052] := 48, [6053] := 48, [6054] := 44, [6055] := 54, [6056] := 46, [6057] := 48, [6058] := 48, [6059] := 48,
        [6060] := 48, [6061] := 48, [6062] := 48, [6063] := 48, [6064] := 48, [6065] := 44, [6066] := 55, [6067] := 46, [6068] := 48, [6069] := 48, [6070] := 48, [6071] := 48, [6072] := 48, [6073] := 48, [6074] := 48, [6075] := 48, [6076] := 44, [6077] := 56, [6078] := 46, [6079] := 48, [6080] := 48, [6081] := 48, [6082] := 48, [6083] := 48, [6084] := 48, [6085] := 48, [6086] := 48, [6087] := 44, [6088] := 57, [6089] := 46, [6090] := 48, [6091] := 48, [6092] := 48, [6093] := 48, [6094] := 48, [6095] := 48, [6096] := 48, [6097] := 48, [6098] := 44, [6099] := 49, [6100] := 48, [6101] := 46, [6102] := 48, [6103] := 48, [6104] := 48, [6105] := 48, [6106] := 48, [6107] := 48, [6108] := 48, [6109] := 44, [6110] := 49, [6111] := 49, [6112] := 46, [6113] := 48, [6114] := 48, [6115] := 48, [6116] := 48, [6117] := 48, [6118] := 48, [6119] := 48,
        [6120] := 44, [6121] := 49, [6122] := 50, [6123] := 46, [6124] := 48, [6125] := 48, [6126] := 48, [6127] := 48, [6128] := 48, [6129] := 48, [6130] := 48, [6131] := 44, [6132] := 49, [6133] := 46, [6134] := 48, [6135] := 48, [6136] := 48, [6137] := 48, [6138] := 48, [6139] := 48, [6140] := 48, [6141] := 48, [6142] := 13, [6143] := 10, [6144] := 51, [6145] := 53, [6146] := 56, [6147] := 56, [6148] := 56, [6149] := 44, [6150] := 48, [6151] := 46, [6152] := 48, [6153] := 57, [6154] := 51, [6155] := 50, [6156] := 54, [6157] := 50, [6158] := 49, [6159] := 53, [6160] := 44, [6161] := 50, [6162] := 46, [6163] := 48, [6164] := 48, [6165] := 48, [6166] := 48, [6167] := 48, [6168] := 48, [6169] := 48, [6170] := 48, [6171] := 44, [6172] := 53, [6173] := 46, [6174] := 48, [6175] := 48, [6176] := 48, [6177] := 48, [6178] := 48, [6179] := 48,
        [6180] := 48, [6181] := 48, [6182] := 44, [6183] := 54, [6184] := 46, [6185] := 48, [6186] := 48, [6187] := 48, [6188] := 48, [6189] := 48, [6190] := 48, [6191] := 48, [6192] := 48, [6193] := 44, [6194] := 55, [6195] := 46, [6196] := 48, [6197] := 48, [6198] := 48, [6199] := 48, [6200] := 48, [6201] := 48, [6202] := 48, [6203] := 48, [6204] := 44, [6205] := 56, [6206] := 46, [6207] := 48, [6208] := 48, [6209] := 48, [6210] := 48, [6211] := 48, [6212] := 48, [6213] := 48, [6214] := 48, [6215] := 44, [6216] := 57, [6217] := 46, [6218] := 48, [6219] := 48, [6220] := 48, [6221] := 48, [6222] := 48, [6223] := 48, [6224] := 48, [6225] := 48, [6226] := 44, [6227] := 49, [6228] := 48, [6229] := 46, [6230] := 48, [6231] := 48, [6232] := 48, [6233] := 48, [6234] := 48, [6235] := 48, [6236] := 48, [6237] := 44, [6238] := 49, [6239] := 49,
        [6240] := 46, [6241] := 48, [6242] := 48, [6243] := 48, [6244] := 48, [6245] := 48, [6246] := 48, [6247] := 48, [6248] := 44, [6249] := 49, [6250] := 50, [6251] := 46, [6252] := 48, [6253] := 48, [6254] := 48, [6255] := 48, [6256] := 48, [6257] := 48, [6258] := 48, [6259] := 44, [6260] := 49, [6261] := 46, [6262] := 48, [6263] := 48, [6264] := 48, [6265] := 48, [6266] := 48, [6267] := 48, [6268] := 48, [6269] := 48, [6270] := 13, [6271] := 10, [6272] := 51, [6273] := 53, [6274] := 56, [6275] := 56, [6276] := 56, [6277] := 44, [6278] := 48, [6279] := 46, [6280] := 48, [6281] := 57, [6282] := 51, [6283] := 50, [6284] := 55, [6285] := 51, [6286] := 55, [6287] := 51, [6288] := 44, [6289] := 50, [6290] := 46, [6291] := 48, [6292] := 48, [6293] := 48, [6294] := 48, [6295] := 48, [6296] := 48, [6297] := 48, [6298] := 48, [6299] := 44,
        [6300] := 53, [6301] := 46, [6302] := 48, [6303] := 48, [6304] := 48, [6305] := 48, [6306] := 48, [6307] := 48, [6308] := 48, [6309] := 48, [6310] := 44, [6311] := 54, [6312] := 46, [6313] := 48, [6314] := 48, [6315] := 48, [6316] := 48, [6317] := 48, [6318] := 48, [6319] := 48, [6320] := 48, [6321] := 44, [6322] := 55, [6323] := 46, [6324] := 48, [6325] := 48, [6326] := 48, [6327] := 48, [6328] := 48, [6329] := 48, [6330] := 48, [6331] := 48, [6332] := 44, [6333] := 56, [6334] := 46, [6335] := 48, [6336] := 48, [6337] := 48, [6338] := 48, [6339] := 48, [6340] := 48, [6341] := 48, [6342] := 48, [6343] := 44, [6344] := 57, [6345] := 46, [6346] := 48, [6347] := 48, [6348] := 48, [6349] := 48, [6350] := 48, [6351] := 48, [6352] := 48, [6353] := 48, [6354] := 44, [6355] := 49, [6356] := 48, [6357] := 46, [6358] := 48, [6359] := 48,
        [6360] := 48, [6361] := 48, [6362] := 48, [6363] := 48, [6364] := 48, [6365] := 44, [6366] := 49, [6367] := 49, [6368] := 46, [6369] := 48, [6370] := 48, [6371] := 48, [6372] := 48, [6373] := 48, [6374] := 48, [6375] := 48, [6376] := 44, [6377] := 49, [6378] := 50, [6379] := 46, [6380] := 48, [6381] := 48, [6382] := 48, [6383] := 48, [6384] := 48, [6385] := 48, [6386] := 48, [6387] := 44, [6388] := 49, [6389] := 46, [6390] := 48, [6391] := 48, [6392] := 48, [6393] := 48, [6394] := 48, [6395] := 48, [6396] := 48, [6397] := 48, [6398] := 13, [6399] := 10, [6400] := 51, [6401] := 53, [6402] := 56, [6403] := 56, [6404] := 56, [6405] := 44, [6406] := 48, [6407] := 46, [6408] := 48, [6409] := 57, [6410] := 51, [6411] := 50, [6412] := 56, [6413] := 53, [6414] := 51, [6415] := 49, [6416] := 44, [6417] := 50, [6418] := 46, [6419] := 48,
        [6420] := 48, [6421] := 48, [6422] := 48, [6423] := 48, [6424] := 48, [6425] := 48, [6426] := 48, [6427] := 44, [6428] := 53, [6429] := 46, [6430] := 48, [6431] := 48, [6432] := 48, [6433] := 48, [6434] := 48, [6435] := 48, [6436] := 48, [6437] := 48, [6438] := 44, [6439] := 54, [6440] := 46, [6441] := 48, [6442] := 48, [6443] := 48, [6444] := 48, [6445] := 48, [6446] := 48, [6447] := 48, [6448] := 48, [6449] := 44, [6450] := 55, [6451] := 46, [6452] := 48, [6453] := 48, [6454] := 48, [6455] := 48, [6456] := 48, [6457] := 48, [6458] := 48, [6459] := 48, [6460] := 44, [6461] := 56, [6462] := 46, [6463] := 48, [6464] := 48, [6465] := 48, [6466] := 48, [6467] := 48, [6468] := 48, [6469] := 48, [6470] := 48, [6471] := 44, [6472] := 57, [6473] := 46, [6474] := 48, [6475] := 48, [6476] := 48, [6477] := 48, [6478] := 48, [6479] := 48,
        [6480] := 48, [6481] := 48, [6482] := 44, [6483] := 49, [6484] := 48, [6485] := 46, [6486] := 48, [6487] := 48, [6488] := 48, [6489] := 48, [6490] := 48, [6491] := 48, [6492] := 48, [6493] := 44, [6494] := 49, [6495] := 49, [6496] := 46, [6497] := 48, [6498] := 48, [6499] := 48, [6500] := 48, [6501] := 48, [6502] := 48, [6503] := 48, [6504] := 44, [6505] := 49, [6506] := 50, [6507] := 46, [6508] := 48, [6509] := 48, [6510] := 48, [6511] := 48, [6512] := 48, [6513] := 48, [6514] := 48, [6515] := 44, [6516] := 49, [6517] := 46, [6518] := 48, [6519] := 48, [6520] := 48, [6521] := 48, [6522] := 48, [6523] := 48, [6524] := 48, [6525] := 48, [6526] := 13, [6527] := 10, [6528] := 51, [6529] := 53, [6530] := 56, [6531] := 56, [6532] := 56, [6533] := 44, [6534] := 48, [6535] := 46, [6536] := 48, [6537] := 57, [6538] := 51, [6539] := 50,
        [6540] := 57, [6541] := 54, [6542] := 56, [6543] := 56, [6544] := 44, [6545] := 50, [6546] := 46, [6547] := 48, [6548] := 48, [6549] := 48, [6550] := 48, [6551] := 48, [6552] := 48, [6553] := 48, [6554] := 48, [6555] := 44, [6556] := 53, [6557] := 46, [6558] := 48, [6559] := 48, [6560] := 48, [6561] := 48, [6562] := 48, [6563] := 48, [6564] := 48, [6565] := 48, [6566] := 44, [6567] := 54, [6568] := 46, [6569] := 48, [6570] := 48, [6571] := 48, [6572] := 48, [6573] := 48, [6574] := 48, [6575] := 48, [6576] := 48, [6577] := 44, [6578] := 55, [6579] := 46, [6580] := 48, [6581] := 48, [6582] := 48, [6583] := 48, [6584] := 48, [6585] := 48, [6586] := 48, [6587] := 48, [6588] := 44, [6589] := 56, [6590] := 46, [6591] := 48, [6592] := 48, [6593] := 48, [6594] := 48, [6595] := 48, [6596] := 48, [6597] := 48, [6598] := 48, [6599] := 44,
